// TwinCAT 3 PLC project MPS
// Title: MPS
// Company: Cosylab
// ProjectVersion: 0.1
// ProgramVersion: 3.1.4023.0
// libraries:
//   Tc2_Standard, * (Beckhoff Automation GmbH)
//   Tc2_System, * (Beckhoff Automation GmbH)
//   Tc3_Module, * (Beckhoff Automation GmbH)
// project tree:
//   DUTs/ E_2PosMonState.TcDUT, E_3PosMonState.TcDUT, E_EpicsMeasurementState.TcDUT, E_KlystronState.TcDUT, E_KlystronPPSState.TcDUT, E_MpsFault.TcDUT, E_MpsFaultSeverity.TcDUT, E_MpsState.TcDUT, E_MpsWarning.TcDUT
//   / GlobalTextList.TcGTLO, PlcTask.TcTTO, Visualization Manager.TcVMO (not stored)
//   GVLs/ CONSTANTS.TcGVL, G_EPICS.TcGVL, IO.TcGVL
//   GVLs/EpicsInterfaceDef/ ST_FaultList.TcDUT, ST_FlowMeter.TcDUT, ST_InterlockOutput.TcDUT, ST_EpicsMeasurement.TcDUT, ST_PPSInput.TcDUT, ST_StateController.TcDUT, ST_StateOutput.TcDUT, ST_TwoAxisProfileMonitor.TcDUT, ST_WarningList.TcDUT, ST_TwoAxisPopIn.TcDUT, ST_FastGateValveMonitor.TcDUT, ST_General.TcDUT, ST_LatchingAND.TcDUT, ST_Pressure.TcDUT, ST_RepetitionRate.TcDUT, ST_RtdTemperature.TcDUT, ST_ThreePositionPopIn.TcDUT, ST_TwoPositionPopIn.TcDUT
//   POUs/ FB_FlowMeter.TcPOU, FB_TwoAxisPopIn.TcPOU, FB_EpicsMeasurement.TcPOU, MpsLogicTest.TcPOU, FB_Pressure.TcPOU, FB_StateController.TcPOU, FB_TwoAxisProfileMonitor.TcPOU, FB_TwoPositionPopIn.TcPOU, FB_FastGateValveMonitor.TcPOU, FB_LatchingAND.TcPOU, FB_RepetitionRate.TcPOU, FB_ThreePositionPopIn.TcPOU, FB_Pt100.TcPOU, MAIN.TcPOU, MpsLogic.TcPOU, MpsLogicUpgrade.TcPOU, RtdReadings.TcPOU
//   VISUs/ TestGUI.TcVIS

CONFIGURATION MPS
    RESOURCE PLC ON TwinCAT3
        TASK PlcTask(INTERVAL := T#10ms, PRIORITY := 20);
        PROGRAM MAIN WITH PlcTask : MAIN;
    END_RESOURCE
END_CONFIGURATION

// ---- DUTs/E_2PosMonState.TcDUT
{attribute 'qualified_only'}
{attribute 'strict'}
TYPE E_2PosMonState :
(
	Nan := 0,
	isINSERTED := 1,
	isRETRACTED := 2,
	isMOVING := 3,
	isBROKEN := 4,
	isForcedOut := 5
);
END_TYPE

// ---- DUTs/E_3PosMonState.TcDUT
{attribute 'qualified_only'}
{attribute 'strict'}
TYPE E_3PosMonState :
(
	Nan := 0,
	isINSERTED1 := 1,
	isINSERTED2 := 2,
	isRETRACTED := 3,
	isMOVING := 4,
	isBROKEN := 5,
	isForcedOut := 6
);
END_TYPE

// ---- DUTs/E_EpicsMeasurementState.TcDUT
{attribute 'qualified_only'}
{attribute 'strict'}
TYPE E_EpicsMeasurementState :
(
	Nan := 0,
	isOkay := 1,
	isInactive := 2,
	isOutOfRange := 3,
	hasTimeout := 4
);
END_TYPE

// ---- DUTs/E_KlystronState.TcDUT
{attribute 'qualified_only'}
{attribute 'strict'}
TYPE E_KlystronState :
(
	Off := 1,
	StandbyOffRequested := 3,
	StamdbyOnRequested := 4,
	Standby := 5,
	HVOffRequested := 7,
	HVOnRequested := 8,
	HV := 9,
	TrigOffRequested := 11,
	TrigOnRequested := 12,
	Trig := 13
);
END_TYPE

// ---- DUTs/E_KlystronPPSState.TcDUT
{attribute 'qualified_only'}
{attribute 'strict'}
TYPE E_KlystronPPSState :
(
	Off := 0,
	StandbyMode := 1,
	HVMode := 2,
	TrigMode := 3,
	NoSignal := 4
);
END_TYPE

// ---- DUTs/E_MpsFault.TcDUT
{attribute 'qualified_only'}
{attribute 'strict'}
TYPE E_MpsFault :
(
	NoFault := 0,
	StandbyPPSInterlock := 10,
	StandbyMPSInterlock := 11,
	HVPPSInterlock := 20,
	HVPressureInterlock := 21,
	HVDipoleFlowInterlock := 22,
	HVDipoleThermalInterlock := 23,
	HVRFNetwork02FlowInterlock := 24,
	RFPPSInterlock := 30,
	RFMPSInterlock := 31,
	BeamSolenoidFlowInterlock := 40,
	BeamSolenoidThermalInterock := 41,
	BeamGunFlowInterlock := 42,
	BeamRFNetwork01FlowInterlock := 43,
	BeamPopInInterlock := 44
);
END_TYPE

// ---- DUTs/E_MpsFaultSeverity.TcDUT
{attribute 'qualified_only'}
{attribute 'strict'}
TYPE E_MpsFaultSeverity :
(
	NoFault := 0,
	StandbyFault := 1,
	HVFault := 2,
	RFFault := 3,
	BeamFault := 4
);
END_TYPE

// ---- DUTs/E_MpsState.TcDUT
{attribute 'qualified_only'}
{attribute 'strict'}
TYPE E_MpsState :
(
	OFF := 0,
	ExitingStandby := 1,
	EnteringStandby := 2,
	STANDBY := 3,
	ExitingHV := 4,
	EnteringHV := 5,
	HV := 6,
	SafeRoutine := 7,
	EnteringManualMode := 8,
	ManualMode := 9,
	EnteringAutomaticMode := 10,
	AutomaticMode := 11,
	SelectingEnergySetpoint := 12,
	ApplyingEnergyProfile := 13,
	LowRepRateBeamOn := 14,
	FullBeamOn := 15
);
END_TYPE

// ---- DUTs/E_MpsWarning.TcDUT
{attribute 'qualified_only'}
{attribute 'strict'}
TYPE E_MpsWarning :
(
	NoWarning := 0,
	InvalidStateRequested := 1,
	ManualModeUnreachable := 2,
	AutomaticModeUnreachable := 3
);
END_TYPE

// ---- GVLs/EpicsInterfaceDef/ST_FaultList.TcDUT
TYPE ST_FaultList :
STRUCT
	Fault_1St : E_MpsFault;
	Fault_2St : E_MpsFault;
	Fault_3St : E_MpsFault;
	Fault_4St : E_MpsFault; 
	Fault_5St : E_MpsFault; 
	Fault_6St : E_MpsFault;
	Fault_7St : E_MpsFault;
	Fault_8St : E_MpsFault;
	Fault_9St : E_MpsFault;
	Fault_10St : E_MpsFault;
END_STRUCT
END_TYPE

// ---- GVLs/EpicsInterfaceDef/ST_FlowMeter.TcDUT
TYPE ST_FlowMeter :
STRUCT
	FlowInterlockSt : BOOL;
	TemperatureInterlockSt : BOOL;
	FlowSt : LREAL;
	TemperatureSt : LREAL;
END_STRUCT
END_TYPE

// ---- GVLs/EpicsInterfaceDef/ST_InterlockOutput.TcDUT
TYPE ST_InterlockOutput :
STRUCT
	HPI_SHUTR01_OPEN_OUT : BOOL;
	HPI_SHUTR02_OPEN_OUT : BOOL;
	HPI_SOLN01_ENABLE_OUT : BOOL;
	HPI_DIP01_ENABLE_OUT : BOOL;
	HPI_KLY01_STANDBY_OUT : BOOL;
	HPI_KLY01_HVMODE_OUT : BOOL;
	HPI_KLY01_TRIGMODE_OUT : BOOL;
	HPI_KLY02_STANDBY_OUT : BOOL;
	HPI_KLY02_HVMODE_OUT : BOOL;
	HPI_KLY02_TRIGMODE_OUT : BOOL;
	
	
END_STRUCT
END_TYPE

// ---- GVLs/EpicsInterfaceDef/ST_EpicsMeasurement.TcDUT
TYPE ST_EpicsMeasurement :
STRUCT
	MeasurementValueSt : LREAL := CONSTANTS.MINIMUM_LREAL;
	MeasurementLowThresholdSt : LREAL := CONSTANTS.MINIMUM_LREAL;
	MeasurementHighThresholdSt : LREAL := CONSTANTS.MINIMUM_LREAL;
	InterlockSt : BOOL;
END_STRUCT
END_TYPE

// ---- GVLs/EpicsInterfaceDef/ST_PPSInput.TcDUT
TYPE ST_PPSInput :
STRUCT
	EnableFB_IN : BOOL;
	AllowFB_IN : BOOL;
	RFPowerFB_IN : BOOL;
	
	
END_STRUCT
END_TYPE

// ---- GVLs/EpicsInterfaceDef/ST_StateController.TcDUT
TYPE ST_StateController :
STRUCT
	StateSt : E_MpsState;
	EpicsStateSt : E_MpsState;
	TargetStateEpicsSt : E_MpsState;
	TargetStateSt : E_MpsState;
	
	Klystron01CCPSVolt01St : LREAL;
	Klystron01CCPSVolt02St : LREAL;
	Klystron01StateSt : E_KlystronState;
	Klystron01PPSStateSt : E_KlystronPPSState;
	
	Klystron02CCPSVolt01St : LREAL;
	Klystron02CCPSVolt02St : LREAL;
	Klystron02StateSt : E_KlystronState;
	Klystron02PPSStateSt : E_KlystronPPSState;
	
	FaultSeveritySt : E_MpsFaultSeverity;
	SetTargetStateSt : BOOL;
	ManualModeSt : BOOL;
	AutomaticModeSt : BOOL;
	AllowEnergyProfileLoadSt : BOOL;
	AllowLowRepRateBeamOnSt : BOOL;
	AllowFullBeamOnSt : BOOL;
END_STRUCT
END_TYPE

// ---- GVLs/EpicsInterfaceDef/ST_StateOutput.TcDUT
TYPE ST_StateOutput :
STRUCT
	StandbyEnabled_OUT : BOOL;
	HVEnabled_OUT : BOOL;
	BeamEnabled_OUT : BOOL;
	ManualModeEnabled_OUT : BOOL;
	AutomaticModeEnabled_OUT : BOOL;
END_STRUCT
END_TYPE

// ---- GVLs/EpicsInterfaceDef/ST_TwoAxisProfileMonitor.TcDUT
TYPE ST_TwoAxisProfileMonitor :
STRUCT
	//Controls
	InsertAxis1Cmd : BOOL;
	InsertAxis2Cmd : BOOL;
	RetractCmd : BOOL;
	
	//Statuses
	InsertedAxis1St : BOOL;
	InsertedAxis2St : BOOL;
	RetractedSt : BOOL;
	
	InterlockSt :BOOL;
	
	StateSt : E_3PosMonState;
	
	DisableButtonsSt :BOOL;
		
END_STRUCT
END_TYPE

// ---- GVLs/EpicsInterfaceDef/ST_WarningList.TcDUT
TYPE ST_WarningList :
STRUCT
	Warning_1St : E_MpsWarning;
	Warning_2St : E_MpsWarning;
	Warning_3St : E_MpsWarning;
	Warning_4St : E_MpsWarning; 
	Warning_5St : E_MpsWarning; 
	Warning_6St : E_MpsWarning;
	Warning_7St : E_MpsWarning;
	Warning_8St : E_MpsWarning;
	Warning_9St : E_MpsWarning;
	Warning_10St : E_MpsWarning;
END_STRUCT
END_TYPE

// ---- GVLs/EpicsInterfaceDef/ST_TwoAxisPopIn.TcDUT
TYPE ST_TwoAxisPopIn :
STRUCT
	//Controls
	Axis1_InsertPos2Cmd :BOOL;
	Axis1_RetractPos1Cmd : BOOL;
	
	Axis2_InsertPos2Cmd: BOOL;
	Axis2_RetractPos1Cmd : BOOL;
	
	//Statuses
	
	Axis1_IsInsertedPos2St : BOOL;
	Axis1_IsRetractedPos1St : BOOL;
	
	Axis2_IsInsertedPos2St : BOOL;
	Axis2_IsRetractedPos1St : BOOL;
	
	InterlockSt : BOOL;
	
	Axis1StateSt : E_2PosMonState;
	Axis2StateSt : E_2PosMonState;
	
	DisableButtonsSt :BOOL;
	
END_STRUCT
END_TYPE

// ---- GVLs/EpicsInterfaceDef/ST_FastGateValveMonitor.TcDUT
TYPE ST_FastGateValveMonitor :
STRUCT
	ClosedSt : BOOL;
	OpenSt : BOOL;
	InterlockSt : BOOL;
END_STRUCT
END_TYPE

// ---- GVLs/EpicsInterfaceDef/ST_General.TcDUT
TYPE ST_General :
STRUCT
	AcknowledgeAllCmd : BOOL;
	
END_STRUCT
END_TYPE

// ---- GVLs/EpicsInterfaceDef/ST_LatchingAND.TcDUT
TYPE ST_LatchingAND :
STRUCT
	IN_1St : BOOL;
	IN_2St : BOOL;
	IN_3St : BOOL;
	IN_4St : BOOL; 
	IN_5St : BOOL; 
	IN_6St : BOOL;
	IN_7St : BOOL;
	IN_8St : BOOL;
	IN_9St : BOOL;
	IN_10St : BOOL;
	InterlockSt : BOOL;
END_STRUCT
END_TYPE

// ---- GVLs/EpicsInterfaceDef/ST_Pressure.TcDUT
TYPE ST_Pressure :
STRUCT
	IN_1St : BOOL;
	IN_2St : BOOL;
	InterlockSt : BOOL;
END_STRUCT
END_TYPE

// ---- GVLs/EpicsInterfaceDef/ST_RepetitionRate.TcDUT
TYPE ST_RepetitionRate :
STRUCT
	RepRateAboveThresholdSt : BOOL;
	RepetitionRateHzSt : REAL;
	RepetitionRateHzThreshold : REAL;
END_STRUCT
END_TYPE

// ---- GVLs/EpicsInterfaceDef/ST_RtdTemperature.TcDUT
TYPE ST_RtdTemperature :
STRUCT
	TBL_RTD01_TEMP : REAL;
	TBL_RTD02_TEMP : REAL;
	TBL_RTD03_TEMP : REAL;
	TBL_RTD04_TEMP : REAL;
	TBL_RTD05_TEMP : REAL;
	TBL_RTD06_TEMP : REAL;
END_STRUCT
END_TYPE

// ---- GVLs/EpicsInterfaceDef/ST_ThreePositionPopIn.TcDUT
TYPE ST_ThreePositionPopIn :
STRUCT
	//Controls
	RetractPos1Cmd : BOOL;
	InsertPos2Cmd : BOOL;
	InsertPos3Cmd : BOOL;
	
	//Statuses
	RetractedPos1St : BOOL;
	InsertedPos2St : BOOL;
	InsertedPos3St : BOOL;
	
	InterlockSt :BOOL;
	
	StateSt : E_3PosMonState;
	
	DisableButtonsSt :BOOL;
		
END_STRUCT
END_TYPE

// ---- GVLs/EpicsInterfaceDef/ST_TwoPositionPopIn.TcDUT
TYPE ST_TwoPositionPopIn :
STRUCT
	//Controls
	InsertPos2Cmd : BOOL;
	RetractPos1Cmd : BOOL;
	
	//Statuses
	InsertedPos2St : BOOL;
	RetractedPos1St : BOOL;
	
	InterlockSt :BOOL;
	
	StateSt : E_2PosMonState;
		
END_STRUCT
END_TYPE

// ---- GVLs/CONSTANTS.TcGVL
{attribute 'qualified_only'}
VAR_GLOBAL CONSTANT
	MINIMUM_LREAL : LREAL := -1.7976931348623157E+308;
	MINIMUM_LREAL_THRESHOLD : LREAL := -1.7976931348623157E+300;
	APPROXIMATE_ZERO : LREAL := 0.01;
	MAX_NUMBER_OF_FAULTS : UINT := 10;
	MAX_NUMBER_OF_WARNINGS : UINT := 10;
END_VAR

// ---- GVLs/G_EPICS.TcGVL
{attribute 'qualified_only'}
VAR_GLOBAL

	RepetitionRate : ST_RepetitionRate;	
	
	StateController : ST_StateController;
	StateOutput : ST_StateOutput;

	Pressure : ST_Pressure;
	GunFlowSwitches : ST_LatchingAND;
	FastGateValve : ST_FastGateValveMonitor;
	RfNetwork01FlowSwitches : ST_LatchingAND;
	RfNetwork02FlowSwitches : ST_LatchingAND;
	SolenoidFlow : ST_LatchingAND;
	SolenoidThermalSwitches : ST_LatchingAND;
	DipoleThermalSwitches : ST_LatchingAND;
	DipoleFlow : ST_LatchingAND;
	MagnetField : ST_EpicsMeasurement;
	DipoleCurrent : ST_EpicsMeasurement; 
	
	PopIn01 : ST_ThreePositionPopIn;
	PopIn02 : ST_TwoPositionPopIn;
	PopIn03 : ST_TwoAxisPopIn;
	PopIn04 : ST_ThreePositionPopIn;
	PopIn05 : ST_TwoAxisPopIn;
	PopIn06 : ST_TwoPositionPopIn;
	
	InterlockOutput :ST_InterlockOutput;
	PPSInput : ST_PPSInput;
	
	FaultList : ST_FaultList;
	WarningList : ST_WarningList;
	
	General : ST_General;
	
	RtdTemperature	: ST_RtdTemperature;
	
	Linac1Flow : ST_LatchingAND;
	
	Linac2FlowMeter01 : ST_FlowMeter;
	Linac2FlowMeter02 : ST_FlowMeter;
	Linac2FlowMeter03 : ST_FlowMeter;
	Linac2FlowMeter04 : ST_FlowMeter;
	Linac2FlowMeter05 : ST_FlowMeter;
	Linac2Flow : ST_LatchingAND;
	
END_VAR

// ---- GVLs/IO.TcGVL
{attribute 'qualified_only'}
VAR_GLOBAL
	
BUN1_PULS01_REPRATE_IN   AT %I* : UDINT;   //   Pulse generator repetition rate
BUN1_PULS01_INHIBIT_OUT   AT %Q* : BOOL;   //Pulse generator inhibit
HPI_SHUTR01_OPEN_OUT   AT %Q* : BOOL;   //MPS Shutter, located before the HPI, opens the shutter
HPI_SHUTR02_OPEN_OUT   AT %Q* : BOOL;   //MPS Shutter, located before the HPI, opens the shutter
HPI_VGCC01_PRESSILK_IN   AT %I* : BOOL;   //   Vacuum gauge controller pressure interlock
HPI_IONP01_PRESSILK_IN   AT %I* : BOOL;   //   Ion pump controller pressure interlock
HPI_HPI01_FS1_IN   AT %I* : BOOL;   //   Photoinjector water flow
HPI_HPI01_FS2_IN   AT %I* : BOOL;   //   Photoinjector water flow
HPI_HPI01_FS3_IN   AT %I* : BOOL;   //   Photoinjector water flow
HPI_HPI01_FS4_IN   AT %I* : BOOL;   //   Photoinjector water flow
HPI_HPI01_FS5_IN   AT %I* : BOOL;   //   Photoinjector water flow
HPI_HPI01_FS6_IN   AT %I* : BOOL;   //   Photoinjector water flow
HPI_RFNET01_FS1_IN   AT %I* : BOOL;   //   RF network (loads and windows) water flow
HPI_RFNET02_FS1_IN   AT %I* : BOOL;   //   RF network (loads and windows) water flow
HPI_RFNET02_FS2_IN   AT %I* : BOOL;   //   RF network (loads and windows) water flow
HPI_RFNET02_FS3_IN   AT %I* : BOOL;   //   RF network (loads and windows) water flow
HPI_SOLN01_FS1_IN   AT %I* : BOOL;   //   Solenoid water flow
HPI_SOLN01_FS2_IN   AT %I* : BOOL;   //   Solenoid water flow
HPI_SOLN01_FS3_IN   AT %I* : BOOL;   //   Solenoid water flow
HPI_VALV01_CLOSED_IN   AT %I* : BOOL;   //   Fast acting gate valve
HPI_VALV01_OPEN_IN   AT %I* : BOOL;   //   Fast acting gate valve
HPI_KLY01_STANDBY_OUT    AT %Q* : BOOL;   //Allow Standby
HPI_KLY01_HVMODE_OUT    AT %Q* : BOOL;   //Allow HV mode
HPI_KLY01_TRIGMODE_OUT    AT %Q* : BOOL;   //Allow Trig mode
HPI_KLY02_STANDBY_OUT    AT %Q* : BOOL;   //Allow Standby
HPI_KLY02_HVMODE_OUT    AT %Q* : BOOL;   //Allow HV mode
HPI_KLY02_TRIGMODE_OUT    AT %Q* : BOOL;   //Allow Trig mode
HPI_SOLN01_ENABLE_OUT   AT %Q* : BOOL;   //Enable Solenoid PSU
HPI_DIP01_ENABLE_OUT   AT %Q* : BOOL;   //Enable Dipole PSU
HPI_SOLN01_TEMPILK1_IN   AT %I* : BOOL;   //   Solenoid thermal cutoff
HPI_SOLN01_TEMPILK2_IN   AT %I* : BOOL;   //   Solenoid thermal cutoff
HPI_SOLN01_TEMPILK3_IN   AT %I* : BOOL;   //   Solenoid thermal cutoff
DUMP_DIP01_TEMPILK1_IN   AT %I* : BOOL;   //   Dipole thermal cutoff

TBL_POPIN01_RETRACTED_POS1_IN	AT %I* : BOOL;   //Pop in 01 retracted position 1
TBL_POPIN01_INSERTED_POS2_IN	AT %I* : BOOL;   //Pop in 01 inserted position 2
TBL_POPIN01_INSERTED_POS3_IN	AT %I* : BOOL;   //Pop in 01 inserted position 3
TBL_POPIN01_INSERT_POS2_OUT	AT %Q* : BOOL;   //Insert position 2
TBL_POPIN01_INSERT_POS3_OUT	AT %Q* : BOOL;   //Insert position 3

TBL_POPIN02_RETRACTED_POS1_IN	AT %I* : BOOL;   //Pop in 02 retracted position 1
TBL_POPIN02_INSERTED_POS2_IN	AT %I* : BOOL;   //Pop in 02 inserted position 2
TBL_POPIN02_INSERT_POS2_OUT	AT %Q* : BOOL;   //Insert position 2

TBL_POPIN03_AX1_RETRACTED_POS1_IN   AT %I* : BOOL;   //   Axis1 slit retracted position 1
TBL_POPIN03_AX1_INSERTED_POS2_IN   AT %I* : BOOL;   //   Axis1 slit inserted position 2
TBL_POPIN03_AX1_INSERT_POS2_OUT   AT %Q* : BOOL;   //Axis1 insert position 2
TBL_POPIN03_AX2_RETRACTED_POS1_IN   AT %I* : BOOL;   //   Axis2 slit retracted 1
TBL_POPIN03_AX2_INSERTED_POS2_IN   AT %I* : BOOL;   //   Axis2 slit inserted 2
TBL_POPIN03_AX2_INSERT_POS2_OUT   AT %Q* : BOOL;   //Axis2 insert position 2

TBL_POPIN04_RETRACTED_POS1_IN	AT %I* : BOOL;   //Pop in 04 retracted position 1
TBL_POPIN04_INSERTED_POS2_IN	AT %I* : BOOL;   //Pop in 04 inserted position 2
TBL_POPIN04_INSERTED_POS3_IN	AT %I* : BOOL;   //Pop in 04 inserted position 3
TBL_POPIN04_INSERT_POS2_OUT	AT %Q* : BOOL;   //Insert position 2
TBL_POPIN04_INSERT_POS3_OUT	AT %Q* : BOOL;   //Insert position 3

TBL_POPIN05_AX1_RETRACTED_POS1_IN   AT %I* : BOOL;   //   Axis1 slit retracted position 1
TBL_POPIN05_AX1_INSERTED_POS2_IN   AT %I* : BOOL;  //   Axis1 slit inserted position 2
TBL_POPIN05_AX1_INSERT_POS2_OUT   AT %Q* : BOOL;   //Axis1 insert position 2
TBL_POPIN05_AX2_RETRACTED_POS1_IN   AT %I* : BOOL;   //   Axis2 slit retracted 1
TBL_POPIN05_AX2_INSERTED_POS2_IN   AT %I* : BOOL;   //   Axis2 slit inserted 2
TBL_POPIN05_AX2_INSERT_POS2_OUT   AT %Q* : BOOL;   //Axis2 insert position 2

TBL_POPIN06_RETRACTED_POS1_IN	AT %I* : BOOL;   //Pop in 06 retracted position 1
TBL_POPIN06_INSERTED_POS2_IN	AT %I* : BOOL;   //Pop in 06 inserted position 2
TBL_POPIN06_INSERT_POS2_OUT	AT %Q* : BOOL;   //Insert position 2


LIN1_FS1_IN  AT %I* : BOOL;   //   Linac 1 water flow
LIN1_FS2_IN  AT %I* : BOOL;   //   Linac 1 water flow
LIN1_FS3_IN  AT %I* : BOOL;   //   Linac 1 water flow
LIN1_FS4_IN  AT %I* : BOOL;   //   Linac 1 water flow


TBL_RTD01_TEMP   AT %I* : INT;   //   RTD temperature sensor
TBL_RTD02_TEMP   AT %I* : INT;   //   RTD temperature sensor
TBL_RTD03_TEMP   AT %I* : INT;   //   RTD temperature sensor
TBL_RTD04_TEMP   AT %I* : INT;   //   RTD temperature sensor
TBL_RTD05_TEMP   AT %I* : INT;   //   RTD temperature sensor
TBL_RTD06_TEMP   AT %I* : INT;   //   RTD temperature sensor

BUN1_IOLINK_CH01_IN AT %I* : ARRAY[0..7] OF BYTE;
BUN1_IOLINK_CH02_IN AT %I* : ARRAY[0..7] OF BYTE;
BUN1_IOLINK_CH03_IN AT %I* : ARRAY[0..7] OF BYTE;
BUN1_IOLINK_CH04_IN AT %I* : ARRAY[0..7] OF BYTE;
BUN1_IOLINK_CH05_IN AT %I* : ARRAY[0..7] OF BYTE;
BUN1_IOLINK_CH06_IN AT %I* : ARRAY[0..7] OF BYTE;



END_VAR

// ---- POUs/MAIN.TcPOU
PROGRAM MAIN
VAR
	MpsLogicUpgrade : MpsLogicUpgrade;
	RtdReadings : RtdReadings;
	//MpsLogicTest : MpsLogicTest;
	
END_VAR

//EPICS test

MpsLogicUpgrade();
RtdReadings();

//MpsLogicTest();

END_PROGRAM

// ---- POUs/MpsLogicUpgrade.TcPOU
FUNCTION_BLOCK MpsLogicUpgrade

VAR
	RepetitionRate : FB_RepetitionRate;	

	StateController : FB_StateController;
	StandbyEnabled : BOOL;
	HVEnabled : BOOL;
	HVRampDown : BOOL;
	BeamEnabled : BOOL;
	BeamRampDown : BOOL;
	ManualModeEnabled : BOOL;
	AutomaticModeEnabled : BOOL;
	
	//Interlock conditions
	StandbyInterlock :  BOOL;
	HVInterlock : BOOL;
	RFInterlock : BOOL;
	BeamInterlock : BOOL;
	
	Pressure : FB_Pressure;
	GunFlowSwitches : FB_LatchingAND;
	FastGateValve : FB_FastGateValveMonitor;
	RfNetwork01FlowSwitches : FB_LatchingAND;
	RfNetwork02FlowSwitches : FB_LatchingAND;
	SolenoidFlow : FB_LatchingAND;
	SolenoidThermalSwitches : FB_LatchingAND;
	DipoleThermalSwitches : FB_LatchingAND;
	DipoleFlow : FB_LatchingAND;
	DipoleCurrent : FB_EpicsMeasurement;
	MagnetField : FB_EpicsMeasurement;
	
	PopIn01 : FB_ThreePositionPopIn;
	PopIn02 : FB_TwoPositionPopIn;
	PopIn03 : FB_TwoAxisPopIn;
	PopIn04 : FB_ThreePositionPopIn;
	PopIn05 : FB_TwoAxisPopIn;
	PopIn06 : FB_TwoPositionPopIn;
	
	Linac1Flow : FB_LatchingAND;
	
	Linac2FlowMeter01 : FB_FlowMeter;
	Linac2FlowMeter02 : FB_FlowMeter;
	Linac2FlowMeter03 : FB_FlowMeter;
	Linac2FlowMeter04 : FB_FlowMeter;
	Linac2FlowMeter05 : FB_FlowMeter;
	Linac2Flow : FB_LatchingAND;
	
END_VAR

// Acknowledge interlocks for the FB that needs it
IF G_Epics.General.AcknowledgeAllCmd THEN
	G_Epics.General.AcknowledgeAllCmd := FALSE;
	StateController.Acknowledge();
	GunFlowSwitches.Acknowledge();
	RfNetwork01FlowSwitches.Acknowledge();
	RfNetwork02FlowSwitches.Acknowledge();
	SolenoidThermalSwitches.Acknowledge();
	DipoleThermalSwitches.Acknowledge();
	SolenoidFlow.Acknowledge();
	DipoleFlow.Acknowledge();
	DipoleCurrent.Acknowledge();
	MagnetField.Acknowledge();
	Linac1Flow.Acknowledge();
	Linac2Flow.Acknowledge();
END_IF

//======================== EPICS exchange of data =======================
StateController.Control(structure := G_Epics.StateController);

RepetitionRate.Control(structure:=G_Epics.RepetitionRate);
Pressure.Control(structure:=G_Epics.Pressure);
GunFlowSwitches.Control(structure:=G_Epics.GunFlowSwitches);
FastGateValve.Control(structure:=G_Epics.FastGateValve);
RfNetwork01FlowSwitches.Control(structure:=G_Epics.RfNetwork01FlowSwitches);
RfNetwork02FlowSwitches.Control(structure:=G_Epics.RfNetwork02FlowSwitches);
SolenoidFlow.Control(structure:=G_Epics.SolenoidFlow);
SolenoidThermalSwitches.Control(structure:=G_Epics.SolenoidThermalSwitches);
DipoleThermalSwitches.Control(structure:=G_Epics.DipoleThermalSwitches);
DipoleFlow.Control(structure:=G_Epics.DipoleFlow);
DipoleCurrent.Control(structure:=G_Epics.DipoleCurrent);
MagnetField.Control(structure:=G_Epics.MagnetField);
Linac1Flow.Control(structure:=G_Epics.Linac1Flow);
Linac2Flow.Control(structure:=G_Epics.Linac2Flow);
	

PopIn01.Control(structure:=G_Epics.PopIn01);
PopIn02.Control(structure:=G_Epics.PopIn02);
PopIn03.Control(structure:=G_Epics.PopIn03);
PopIn04.Control(structure:=G_Epics.PopIn04);
PopIn05.Control(structure:=G_Epics.PopIn05);
PopIn06.Control(structure:=G_Epics.PopIn06);

Linac2FlowMeter01.Control(structure := G_EPICS.Linac2FlowMeter01);
Linac2FlowMeter02.Control(structure := G_EPICS.Linac2FlowMeter02);
Linac2FlowMeter03.Control(structure := G_EPICS.Linac2FlowMeter03);
Linac2FlowMeter04.Control(structure := G_EPICS.Linac2FlowMeter04);
Linac2FlowMeter05.Control(structure := G_EPICS.Linac2FlowMeter05);

//Transfer interlock outputs
G_EPICS.InterlockOutput.HPI_KLY01_STANDBY_OUT:=IO.HPI_KLY01_STANDBY_OUT;
G_EPICS.InterlockOutput.HPI_KLY01_HVMODE_OUT:=IO.HPI_KLY01_HVMODE_OUT;
G_EPICS.InterlockOutput.HPI_KLY01_TRIGMODE_OUT:=IO.HPI_KLY01_TRIGMODE_OUT;
G_EPICS.InterlockOutput.HPI_KLY02_STANDBY_OUT:=IO.HPI_KLY02_STANDBY_OUT;
G_EPICS.InterlockOutput.HPI_KLY02_HVMODE_OUT:=IO.HPI_KLY02_HVMODE_OUT;
G_EPICS.InterlockOutput.HPI_KLY02_TRIGMODE_OUT:=IO.HPI_KLY02_TRIGMODE_OUT;
G_EPICS.InterlockOutput.HPI_SHUTR01_OPEN_OUT:=IO.HPI_SHUTR01_OPEN_OUT;
G_EPICS.InterlockOutput.HPI_SHUTR02_OPEN_OUT:=IO.HPI_SHUTR02_OPEN_OUT;
G_EPICS.InterlockOutput.HPI_SOLN01_ENABLE_OUT:=IO.HPI_SOLN01_ENABLE_OUT;
G_EPICS.InterlockOutput.HPI_DIP01_ENABLE_OUT:=IO.HPI_DIP01_ENABLE_OUT;

//Transfer state information
G_EPICS.StateOutput.StandbyEnabled_OUT := StandbyEnabled;
G_EPICS.StateOutput.HVEnabled_OUT := HVEnabled;
G_EPICS.StateOutput.BeamEnabled_OUT := BeamEnabled;
G_EPICS.StateOutput.ManualModeEnabled_OUT := ManualModeEnabled;
G_EPICS.StateOutput.AutomaticModeEnabled_OUT := AutomaticModeEnabled;

//Transfer faults and warnings
G_EPICS.FaultList.Fault_1St := StateController.Fault_OUT[0];
G_EPICS.FaultList.Fault_2St := StateController.Fault_OUT[1];
G_EPICS.FaultList.Fault_3St := StateController.Fault_OUT[2];
G_EPICS.FaultList.Fault_4St := StateController.Fault_OUT[3];
G_EPICS.FaultList.Fault_5St := StateController.Fault_OUT[4];
G_EPICS.FaultList.Fault_6St := StateController.Fault_OUT[5];
G_EPICS.FaultList.Fault_7St := StateController.Fault_OUT[6];
G_EPICS.FaultList.Fault_8St := StateController.Fault_OUT[7];
G_EPICS.FaultList.Fault_9St := StateController.Fault_OUT[8];
G_EPICS.FaultList.Fault_10St := StateController.Fault_OUT[9];

G_EPICS.WarningList.Warning_1St := StateController.Warning_OUT[0];
G_EPICS.WarningList.Warning_2St := StateController.Warning_OUT[1];
G_EPICS.WarningList.Warning_3St := StateController.Warning_OUT[2];
G_EPICS.WarningList.Warning_4St := StateController.Warning_OUT[3];
G_EPICS.WarningList.Warning_5St := StateController.Warning_OUT[4];
G_EPICS.WarningList.Warning_6St := StateController.Warning_OUT[5];
G_EPICS.WarningList.Warning_7St := StateController.Warning_OUT[6];
G_EPICS.WarningList.Warning_8St := StateController.Warning_OUT[7];
G_EPICS.WarningList.Warning_9St := StateController.Warning_OUT[8];
G_EPICS.WarningList.Warning_10St := StateController.Warning_OUT[9];

//======================== ELEMENT INSTANCES ======================	

//State controller
StateController(StandbyEnabled_OUT => StandbyEnabled,
				HVEnabled_OUT => HVEnabled,
				HVRampDown_OUT => HVRampDown,
				BeamEnabled_OUT => BeamEnabled,
				BeamRampDown_OUT => BeamRampDown,
				ManualModeEnabled_OUT => ManualModeEnabled,
				AutomaticModeEnabled_OUT => AutomaticModeEnabled);

//Repetition rate calculation and comparison
RepetitionRate(frequencyRaw := IO.BUN1_PULS01_REPRATE_IN, Inhibit => IO.BUN1_PULS01_INHIBIT_OUT);

//Pop ins
PopIn01(RepRate := RepetitionRate.AboveThreshold,
		Retracted_Pos1_IN := IO.TBL_POPIN01_RETRACTED_POS1_IN,
		Inserted_Pos2_IN := IO.TBL_POPIN01_INSERTED_POS2_IN,
		Inserted_Pos3_IN := IO.TBL_POPIN01_INSERTED_POS3_IN,
		Insert_Pos2_OUT => IO.TBL_POPIN01_INSERT_POS2_OUT,
		Insert_Pos3_OUT => IO.TBL_POPIN01_INSERT_POS3_OUT);

PopIn02(RepRate := RepetitionRate.AboveThreshold,
		Retracted_Pos1_IN := IO.TBL_POPIN02_RETRACTED_POS1_IN,
		Inserted_Pos2_IN := IO.TBL_POPIN02_INSERTED_POS2_IN,
		Insert_Pos2_OUT => IO.TBL_POPIN02_INSERT_POS2_OUT);

PopIn03(RepRate:=RepetitionRate.AboveThreshold,
		Axis1_RetractedPos1_IN:=IO.TBL_POPIN03_AX1_RETRACTED_POS1_IN,
		Axis1_InsertedPos2_IN:=IO.TBL_POPIN03_AX1_INSERTED_POS2_IN,
		Axis1_InsertPos2_OUT=>IO.TBL_POPIN03_AX1_INSERT_POS2_OUT,
		Axis2_RetractedPos1_IN:=IO.TBL_POPIN03_AX2_RETRACTED_POS1_IN,
		Axis2_InsertedPos2_IN:=IO.TBL_POPIN03_AX2_INSERTED_POS2_IN,
		Axis2_InsertPos2_OUT=>IO.TBL_POPIN03_AX2_INSERT_POS2_OUT);

PopIn04(RepRate := RepetitionRate.AboveThreshold,
		Retracted_Pos1_IN := IO.TBL_POPIN04_RETRACTED_POS1_IN,
		Inserted_Pos2_IN := IO.TBL_POPIN04_INSERTED_POS2_IN,
		Inserted_Pos3_IN := IO.TBL_POPIN04_INSERTED_POS3_IN,
		Insert_Pos2_OUT => IO.TBL_POPIN04_INSERT_POS2_OUT,
		Insert_Pos3_OUT => IO.TBL_POPIN04_INSERT_POS3_OUT);
	
PopIn05(RepRate:=RepetitionRate.AboveThreshold,
		Axis1_RetractedPos1_IN:=IO.TBL_POPIN05_AX1_RETRACTED_POS1_IN,
		Axis1_InsertedPos2_IN:=IO.TBL_POPIN05_AX1_INSERTED_POS2_IN,
		Axis1_InsertPos2_OUT=>IO.TBL_POPIN05_AX1_INSERT_POS2_OUT,
		Axis2_RetractedPos1_IN:=IO.TBL_POPIN05_AX2_RETRACTED_POS1_IN,
		Axis2_InsertedPos2_IN:=IO.TBL_POPIN05_AX2_INSERTED_POS2_IN,
		Axis2_InsertPos2_OUT=>IO.TBL_POPIN05_AX2_INSERT_POS2_OUT );				
		
PopIn06(RepRate := RepetitionRate.AboveThreshold,
		Retracted_Pos1_IN := IO.TBL_POPIN06_RETRACTED_POS1_IN,
		Inserted_Pos2_IN := IO.TBL_POPIN06_INSERTED_POS2_IN,
		Insert_Pos2_OUT => IO.TBL_POPIN06_INSERT_POS2_OUT);			

//Pressure interlock
Pressure(IN_1 := IO.HPI_VGCC01_PRESSILK_IN,  IN_2 := IO.HPI_IONP01_PRESSILK_IN);

//Gun flow switches interlock		 
GunFlowSwitches(IN_1 := IO.HPI_HPI01_FS1_IN,
				IN_2 := IO.HPI_HPI01_FS2_IN,
				IN_3 := IO.HPI_HPI01_FS3_IN,
				IN_4 := IO.HPI_HPI01_FS4_IN,
				//IN_5 := IO.HPI_HPI01_FS5_IN,
				IN_6 := IO.HPI_HPI01_FS6_IN );

// RF network, solenoid flow switches...		 
RfNetwork01FlowSwitches(IN_1 := IO.HPI_RFNET01_FS1_IN);
RfNetwork02FlowSwitches(IN_1 := IO.HPI_RFNET02_FS1_IN, IN_2 := IO.HPI_RFNET02_FS2_IN);// IN_3 := IO.HPI_RFNET02_FS3_IN);

SolenoidFlow(IN_1 := IO.HPI_SOLN01_FS1_IN, IN_2 := IO.HPI_SOLN01_FS2_IN, IN_3 := IO.HPI_SOLN01_FS3_IN);

SolenoidThermalSwitches(IN_1:=IO.HPI_SOLN01_TEMPILK1_IN, IN_2:=IO.HPI_SOLN01_TEMPILK2_IN, IN_3:=IO.HPI_SOLN01_TEMPILK3_IN);

DipoleThermalSwitches(IN_1:=IO.DUMP_DIP01_TEMPILK1_IN);

//HPI - Photon injector, TBL - Test beam line
DipoleFlow();//IN_1 := Linac2FlowMeter05.FlowInterlock_OUT);		

DipoleCurrent(InterlockActive_IN:=AutomaticModeEnabled, MeasurementValue_OUT => G_Epics.MagnetField.MeasurementValueSt);
MagnetField(InterlockActive_IN:=AutomaticModeEnabled, MeasurementValue_OUT => G_Epics.MagnetField.MeasurementValueSt);

FastGateValve(Closed:=IO.HPI_VALV01_CLOSED_IN, Open:=IO.HPI_VALV01_OPEN_IN);

Linac1Flow(IN_1 := IO.LIN1_FS1_IN, IN_2 := IO.LIN1_FS2_IN); // IN_3 := IO.LIN1_FS3_IN, IN_4 := IO.LIN1_FS4_IN);

Linac2FlowMeter01(FlowChannel_IN := IO.BUN1_IOLINK_CH06_IN);
Linac2FlowMeter02(FlowChannel_IN := IO.BUN1_IOLINK_CH02_IN);
Linac2FlowMeter03(FlowChannel_IN := IO.BUN1_IOLINK_CH03_IN);
Linac2FlowMeter04(FlowChannel_IN := IO.BUN1_IOLINK_CH04_IN);
Linac2FlowMeter05(FlowChannel_IN := IO.BUN1_IOLINK_CH05_IN);
Linac2Flow(IN_1 := Linac2FlowMeter01.FlowInterlock_OUT, IN_2 := Linac2FlowMeter02.FlowInterlock_OUT);
					  //IN_3 := Linac2FlowMeter03.FlowInterlock_OUT, IN_4 := Linac2FlowMeter04.FlowInterlock_OUT,
					  //IN_5 := Linac2FlowMeter05.FlowInterlock_OUT);

//======================== INTERLOCKS ======================		
//StandbyInterlock := G_EPICS.PPSInput.EnableFB_IN;
StandbyInterlock := G_EPICS.PPSInput.EnableFB_IN;
HVInterlock := StandbyInterlock AND  Pressure.Interlock AND RfNetwork02FlowSwitches.Interlock AND
			DipoleFlow.Interlock AND DipoleThermalSwitches.Interlock AND Linac1Flow.Interlock AND Linac2Flow.Interlock AND
			G_EPICS.PPSInput.AllowFB_IN;
RFInterlock := HVEnabled AND HVInterlock AND 
			G_EPICS.PPSInput.RFPowerFB_IN;
BeamInterlock := RFInterlock AND //FastGateValve.Interlock AND 
			SolenoidFlow.Interlock AND SolenoidThermalSwitches.Interlock AND GunFlowSwitches.Interlock AND
			RfNetwork01FlowSwitches.Interlock AND DipoleCurrent.Interlock AND MagnetField.Interlock;
			//Prof01.Interlock AND Prof02.Interlock AND Prof03.Interlock AND Prof04.Interlock AND Prof05.Interlock AND Prof06.Interlock


//Combining inputs for Shutter Interlock output
IO.HPI_SHUTR01_OPEN_OUT := AutomaticModeEnabled AND BeamInterlock;
IO.HPI_SHUTR02_OPEN_OUT := AutomaticModeEnabled AND BeamInterlock;

//Combining inputs for solenoid and dipole interlock output
IO.HPI_SOLN01_ENABLE_OUT := HVEnabled AND HVInterlock;
IO.HPI_DIP01_ENABLE_OUT := HVEnabled AND HVInterlock;

//Combining inputs for  Klystron interlock outputs
IO.HPI_KLY01_STANDBY_OUT := StandbyInterlock;
//IO.HPI_KLY01_STANDBY_OUT := StandbyEnabled AND StandbyInterlock;
IO.HPI_KLY01_HVMODE_OUT := (AutomaticModeEnabled OR BeamRampDown) AND BeamInterlock;
IO.HPI_KLY01_TRIGMODE_OUT := (AutomaticModeEnabled OR BeamRampDown)AND BeamInterlock;

IO.HPI_KLY02_STANDBY_OUT := StandbyInterlock;
//IO.HPI_KLY02_STANDBY_OUT := StandbyEnabled AND StandbyInterlock;
IO.HPI_KLY02_HVMODE_OUT := (HVEnabled OR HVRampDown) AND HVInterlock;
IO.HPI_KLY02_TRIGMODE_OUT := (ManualModeEnabled OR AutomaticModeEnabled OR BeamRampDown) AND RFInterlock;

IF StandbyEnabled AND NOT StandbyInterlock THEN
	IF NOT  G_EPICS.PPSInput.EnableFB_IN THEN
		StateController.AddFault(E_MpsFault.StandbyPPSInterlock, E_MpsFaultSeverity.StandbyFault);
	ELSE
		StateController.AddFault(E_MpsFault.StandbyMPSInterlock, E_MpsFaultSeverity.StandbyFault);
	END_IF
END_IF

IF HVEnabled AND NOT HVInterlock THEN
	IF NOT  G_EPICS.PPSInput.AllowFB_IN THEN
		StateController.AddFault(E_MpsFault.HVPPSInterlock, E_MpsFaultSeverity.HVFault);
	ELSIF NOT Pressure.Interlock THEN
		StateController.AddFault(E_MpsFault.HVPressureInterlock, E_MpsFaultSeverity.HVFault);
	ELSIF NOT DipoleFlow.Interlock THEN
		StateController.AddFault(E_MpsFault.HVDipoleFlowInterlock, E_MpsFaultSeverity.HVFault);
	ELSIF NOT DipoleThermalSwitches.Interlock THEN
		StateController.AddFault(E_MpsFault.HVDipoleThermalInterlock, E_MpsFaultSeverity.HVFault);
	ELSIF NOT RfNetwork02FlowSwitches.Interlock THEN
		StateController.AddFault(E_MpsFault.HVRFNetwork02FlowInterlock, E_MpsFaultSeverity.HVFault);
	END_IF
END_IF

IF (ManualModeEnabled OR AutomaticModeEnabled) AND NOT RFInterlock THEN
	IF NOT G_EPICS.PPSInput.RFPowerFB_IN THEN
		StateController.AddFault(E_MpsFault.RFPPSInterlock, E_MpsFaultSeverity.RFFault);
	ELSE
		StateController.AddFault(E_MpsFault.RFMPSInterlock, E_MpsFaultSeverity.RFFault);
	END_IF
END_IF

IF AutomaticModeEnabled AND NOT BeamInterlock THEN
	IF NOT SolenoidFlow.Interlock THEN
		StateController.AddFault(E_MpsFault.BeamSolenoidFlowInterlock, E_MpsFaultSeverity.BeamFault);
	ELSIF NOT SolenoidThermalSwitches.Interlock THEN
		StateController.AddFault(E_MpsFault.BeamSolenoidThermalInterock, E_MpsFaultSeverity.BeamFault);
	ELSIF NOT GunFlowSwitches.Interlock THEN
		StateController.AddFault(E_MpsFault.BeamGunFlowInterlock, E_MpsFaultSeverity.BeamFault);
	ELSIF NOT RFNetwork01FlowSwitches.Interlock THEN
		StateController.AddFault(E_MpsFault.BeamRFNetwork01FlowInterlock, E_MpsFaultSeverity.BeamFault);
	ELSE
		StateController.AddFault(E_MpsFault.BeamPopInInterlock, E_MpsFaultSeverity.BeamFault);
	END_IF
END_IF

END_FUNCTION_BLOCK

// ---- POUs/FB_RepetitionRate.TcPOU
FUNCTION_BLOCK FB_RepetitionRate
VAR_INPUT
	frequencyRaw : UDINT;
END_VAR
VAR_OUTPUT
	Inhibit : BOOL;
	AboveThreshold : BOOL;
END_VAR
VAR
	RepetitionRateHz : REAL;
END_VAR
VAR CONSTANT
	ScalingFactor: REAL := 100; // Scaling of raw input frequency
	Threshold : REAL := 10.0; // set this for determening AboveThreshold
END_VAR


//check the card how to scale the input and how to set the frequency in configuration
RepetitionRateHz := UDINT_TO_REAL(frequencyRaw)/ScalingFactor;

AboveThreshold := RepetitionRateHz > Threshold;

METHOD Control : BOOL
VAR_IN_OUT
	structure : ST_RepetitionRate;
END_VAR
structure.RepetitionRateHzSt := RepetitionRateHz;
structure.RepRateAboveThresholdSt := AboveThreshold;
structure.RepetitionRateHzThreshold := Threshold;
END_METHOD

END_FUNCTION_BLOCK

// ---- POUs/FB_StateController.TcPOU
FUNCTION_BLOCK FB_StateController
VAR_INPUT
END_VAR
VAR_OUTPUT
	StandbyEnabled_OUT : BOOL := FALSE;
	HVEnabled_OUT : BOOL := FALSE;
	HVRampDown_OUT : BOOL := FALSE;
	BeamEnabled_OUT : BOOL := FALSE;
	BeamRampDown_OUT : BOOL := FALSE;
	ManualModeEnabled_OUT : BOOL := FALSE;
	AutomaticModeEnabled_OUT : BOOL := FALSE;
	Fault_OUT : ARRAY[0..CONSTANTS.MAX_NUMBER_OF_FAULTS] OF E_MpsFault;
	Warning_OUT : ARRAY[0..CONSTANTS.MAX_NUMBER_OF_FAULTS] OF E_MpsWarning;
	FaultSeverity_OUT : E_MpsFaultSeverity;
	
END_VAR
VAR
	State : E_MpsState;
	TargetState : E_MpsState;
	EpicsState_RB : E_MpsState;
	
	
	NumberOfFaults : UINT := 0;
	NumberOfWarnings : UINT := 0;
	Klystron01CCPSVolt01_RB : LREAL := 0;
	Klystron01CCPSVolt02_RB : LREAL := 0;
	Klystron01State_RB : E_KlystronState;
	Klystron01PPSState_RB : E_KlystronPPSState;
	
	Klystron02State_RB : E_KlystronState;
	Klystron02CCPSVolt01_RB : LREAL := 0;
	Klystron02CCPSVolt02_RB : LREAL := 0;
	Klystron02PPSState_RB : E_KlystronPPSState;
	
	ManualMode_SET : BOOL := FALSE;
	AutomaticMode_SET : BOOL := FALSE;
	AllowEnergyProfileLoad_SET : BOOL := FALSE;
	AllowLowRepRateBeamOn_SET : BOOL := FALSE;
	AllowFullBeamOn_SET : BOOL := FALSE;
	
END_VAR

//Handles state tranistion and configures state outputs
IF State = E_MpsState.OFF THEN
	StandbyEnabled_OUT := FALSE;
	HVEnabled_OUT := FALSE;
	HVRampDown_OUT := FALSE;
	BeamEnabled_OUT := FALSE;
	BeamRampDown_OUT := FALSE;
	ManualModeEnabled_OUT := FALSE;
	AutomaticModeEnabled_OUT := FALSE;
	ManualMode_SET := FALSE;
	AutomaticMode_SET := FALSE;

//When the klystron state in any state above OFF changes to Off or StandbyOff requested
//The system will move to exiting Standby state
//The same applies for the readback of the EPICS state
ELSIF State = E_MpsState.ExitingStandby THEN
	//IF Klystron01State_RB = E_KlystronState.Off AND 
	IF TRUE THEN //Klystron02State_RB = E_KlystronState.Off THEN
		TargetState := E_MpsState.OFF;
		State := E_MpsState.OFF;
	END_IF
	StandbyEnabled_OUT := FALSE;
	HVEnabled_OUT := FALSE;
	HVRampDown_OUT := FALSE;
	BeamEnabled_OUT := FALSE;
	BeamRampDown_OUT := FALSE;
	ManualMode_SET := FALSE;
	AutomaticMode_SET := FALSE;

//Move to standby when the klystrons reach standby
ELSIF State = E_MpsState.EnteringStandby AND FaultSeverity_OUT <> E_MpsFaultSeverity.StandbyFault THEN
	StandbyEnabled_OUT := TRUE;
	IF EpicsState_RB = E_MpsState.STANDBY AND //Klystron01State_RB = E_KlystronState.Standby AND 
	    	Klystron02State_RB = E_KlystronState.Standby THEN
		State := E_MpsState.STANDBY;
	END_IF
	
ELSIF Klystron02State_RB = E_KlystronState.Off OR Klystron02State_RB = E_KlystronState.StandbyOffRequested OR
	  //Klystron01State_RB = E_KlystronState.Off OR Klystron01State_RB = E_KlystronState.StandbyOffRequested
		//OR Klystron01PPSState_RB = E_KlystronPPSState.Off OR Klystron01PPSState_RB = E_KlystronPPSState.NoSignal
		//OR Klystron02PPSState_RB = E_KlystronPPSState.Off OR Klystron02PPSState_RB = E_KlystronPPSState.NoSignal
		//EpicsState_RB = E_MpsState.OFF OR 
		EpicsState_RB = E_MpsState.ExitingStandby OR
		FaultSeverity_OUT = E_MpsFaultSeverity.StandbyFault THEN 	
	State := E_MpsState.ExitingStandby;
	
ELSIF State = E_MpsState.STANDBY THEN
	StandbyEnabled_OUT := TRUE;
	HVEnabled_OUT := FALSE;
	HVRampDown_OUT := FALSE;
	BeamEnabled_OUT := FALSE;
	BeamRampDown_OUT := FALSE;
	ManualMode_SET := FALSE;
	AutomaticMode_SET := FALSE;

//When the klystron state in any state above STANDBY changes to Standby or HV Off
//The system will move to exiting HV state
//The same applies for the readback of the EPICS state
ELSIF State = E_MpsState.ExitingHV THEN
	//IF Klystron01State_RB = E_KlystronState.Standby AND
	IF Klystron02State_RB = E_KlystronState.Standby AND 
		Klystron02CCPSVolt01_RB <= CONSTANTS.APPROXIMATE_ZERO AND Klystron02CCPSVolt02_RB <= CONSTANTS.APPROXIMATE_ZERO THEN
		State := E_MpsState.STANDBY;
		TargetState := E_MpsState.STANDBY;
	END_IF 
	HVEnabled_OUT := FALSE;
	HVRampDown_OUT := TRUE;
	BeamEnabled_OUT := FALSE;
	BeamRampDown_OUT := FALSE;
	ManualMode_SET := FALSE;
	AutomaticMode_SET := FALSE;

//Move to HV when the klystrons reach HV
ELSIF State = E_MpsState.EnteringHV AND FaultSeverity_OUT <> E_MpsFaultSeverity.HVFault THEN
	HVEnabled_OUT := TRUE;
	IF EpicsState_RB = E_MpsState.HV AND //Klystron01State_RB = E_KlystronState.Standby AND
			Klystron02State_RB = E_KlystronState.HV THEN
		State := E_MpsState.HV;
	END_IF

ELSIF Klystron02State_RB = E_KlystronState.Standby OR Klystron02State_RB = E_KlystronState.HVOffRequested
		OR EpicsState_RB = E_MpsState.STANDBY OR EpicsState_RB = E_MpsState.ExitingHV 
		OR FaultSeverity_OUT = E_MpsFaultSeverity.HVFault THEN	
	State := E_MpsState.ExitingHV;	

//Case structure manages transition to higher states
ELSIF State = E_MpsState.HV THEN
	StandbyEnabled_OUT := TRUE;
	HVEnabled_OUT := TRUE;
	HVRampDown_OUT := FALSE;
	BeamEnabled_OUT := FALSE;
	BeamRampDown_OUT := FALSE;
	
	IF ManualMode_SET = TRUE THEN
		State := E_MpsState.EnteringManualMode;
	ELSIF AutomaticMode_SET = TRUE THEN
		State := E_MpsState.EnteringAutomaticMode;
	END_IF

ELSIF State = E_MpsState.EnteringManualMode AND FaultSeverity_OUT <> E_MpsFaultSeverity.RFFault THEN
	IF (ManualMode_SET = FALSE) THEN
		State := E_MpsState.SafeRoutine;
	END_IF
	ManualModeEnabled_OUT := TRUE;
	AutomaticModeEnabled_OUT := FALSE;
	IF EpicsState_RB = E_MpsState.HV AND//Klystron01State_RB = E_KlystronState.Standby AND
			Klystron02State_RB = E_KlystronState.Trig THEN
		State := E_MpsState.ManualMode;
	END_IF
	
ELSIF State = E_MpsState.SafeRoutine THEN
	IF EpicsState_RB = E_MpsState.HV AND Klystron02State_RB = E_KlystronState.HV THEN
		State := E_MpsState.HV;
	END_IF
	BeamEnabled_OUT := FALSE;
	BeamRampDown_OUT := TRUE;
	ManualMode_SET := FALSE;
	AutomaticMode_SET := FALSE;
	ManualModeEnabled_OUT := FALSE;
	AutomaticModeEnabled_OUT := FALSE;
	
ELSIF State = E_MpsState.EnteringAutomaticMode AND FaultSeverity_OUT <> E_MpsFaultSeverity.RFFault THEN	
	IF (AutomaticMode_SET = FALSE) THEN
		State := E_MpsState.SafeRoutine;
	END_IF
	BeamEnabled_OUT := TRUE;
	BeamRampDown_OUT := FALSE;
	ManualModeEnabled_OUT := FALSE;
	AutomaticModeEnabled_OUT := TRUE;
	IF EpicsState_RB = E_MpsState.HV AND Klystron01State_RB = E_KlystronState.Trig
			AND Klystron02State_RB = E_KlystronState.Trig THEN
		State := E_MpsState.AutomaticMode;
	END_IF	

ELSIF Klystron02State_RB = E_KlystronState.HV OR Klystron02State_RB = E_KlystronState.TrigOffRequested
		OR FaultSeverity_OUT = E_MpsFaultSeverity.RFFault OR (ManualMode_SET = FALSE AND AutomaticMode_SET = FALSE) THEN	
	State := E_MpsState.SafeRoutine;	
	
ELSIF State = E_MpsState.ManualMode THEN
	BeamEnabled_OUT := FALSE;
	BeamRampDown_OUT := FALSE;
	ManualModeEnabled_OUT := TRUE;
	AutomaticModeEnabled_OUT := FALSE;
	
ELSIF Klystron01State_RB = E_KlystronState.HV OR Klystron01State_RB = E_KlystronState.TrigOffRequested
		OR Klystron02State_RB = E_KlystronState.HV OR Klystron02State_RB = E_KlystronState.TrigOffRequested
		OR FaultSeverity_OUT = E_MpsFaultSeverity.RFFault THEN	
	State := E_MpsState.SafeRoutine;
	
ELSIF State = E_MpsState.AutomaticMode THEN
	BeamEnabled_OUT := TRUE;
	BeamRampDown_OUT := FALSE;
	ManualModeEnabled_OUT := FALSE;
	AutomaticModeEnabled_OUT := TRUE;
	
END_IF

METHOD Acknowledge : BOOL
VAR_INPUT
END_VAR
VAR
	DefaultFault : ARRAY[0..CONSTANTS.MAX_NUMBER_OF_FAULTS] OF E_MpsFault;
	DefaultWarning : ARRAY[0..CONSTANTS.MAX_NUMBER_OF_WARNINGS] OF E_MpsWarning; 
END_VAR
FaultSeverity_OUT := E_MpsFaultSeverity.NoFault;
Fault_OUT := DefaultFault;
Warning_OUT := DefaultWarning;
NumberOfFaults := 0;
NumberOfWarnings := 0;
END_METHOD

METHOD AddFault : BOOL
VAR_INPUT
	Fault_IN : E_MpsFault;
	FaultType_IN : E_MpsFaultSeverity;
END_VAR
IF NumberOfFaults >= CONSTANTS.MAX_NUMBER_OF_FAULTS THEN
	NumberOfFaults := CONSTANTS.MAX_NUMBER_OF_FAULTS - 1; 
END_IF
Fault_OUT[NumberOfFaults] := Fault_IN;

//System fault severity - severity of the most severe active fault
IF FaultSeverity_OUT = E_MpsFaultSeverity.NoFault THEN
	FaultSeverity_OUT := FaultType_IN;
ELSIF FaultSeverity_OUT = E_MpsFaultSeverity.StandbyFault THEN
	FaultSeverity_OUT := E_MpsFaultSeverity.StandbyFault;
ELSIF FaultSeverity_OUT = E_MpsFaultSeverity.HVFault THEN
	IF FaultType_IN = E_MpsFaultSeverity.StandbyFault THEN
		FaultSeverity_OUT := E_MpsFaultSeverity.StandbyFault;
	END_IF
ELSIF FaultSeverity_OUT = E_MpsFaultSeverity.RFFault THEN
	IF FaultType_IN = E_MpsFaultSeverity.StandbyFault OR FaultType_IN = E_MpsFaultSeverity.HVFault THEN
		FaultSeverity_OUT := FaultType_IN;
	END_IF
ELSIF FaultSeverity_OUT = E_MpsFaultSeverity.BeamFault THEN
	IF FaultType_IN <> E_MpsFaultSeverity.NoFault THEN
		FaultSeverity_OUT := FaultType_IN;
	END_IF 
END_IF

NumberOfFaults := NumberOfFaults + 1;
END_METHOD

METHOD AddWarning : BOOL
VAR_INPUT
	Warning_IN : E_MpsWarning;
END_VAR
IF NumberOfWarnings >= CONSTANTS.MAX_NUMBER_OF_WARNINGS THEN
	NumberOfWarnings := CONSTANTS.MAX_NUMBER_OF_WARNINGS - 1; 
END_IF
Warning_OUT[NumberOfWarnings] := Warning_IN;
NumberOfWarnings := NumberOfWarnings + 1;
END_METHOD

METHOD Control : BOOL
VAR_IN_OUT
	structure : ST_StateController;
END_VAR
structure.StateSt := State;
structure.TargetStateSt := TargetState;
EpicsState_RB := structure.EpicsStateSt;
Klystron01CCPSVolt01_RB := structure.Klystron01CCPSVolt01St;
Klystron01CCPSVolt02_RB := structure.Klystron01CCPSVolt02St;
Klystron01State_RB := structure.Klystron01StateSt;
Klystron01PPSState_RB := structure.Klystron01PPSStateSt;

Klystron02CCPSVolt01_RB := structure.Klystron02CCPSVolt01St;
Klystron02CCPSVolt02_RB := structure.Klystron02CCPSVolt02St;
Klystron02State_RB := structure.Klystron02StateSt;
Klystron02PPSState_RB := structure.Klystron02PPSStateSt;
structure.FaultSeveritySt := FaultSeverity_OUT;
IF ManualMode_SET = TRUE THEN
	ManualMode_SET := structure.ManualModeSt;
	IF structure.AutomaticModeSt = TRUE THEN
		AddWarning(Warning_IN := E_MpsWarning.AutomaticModeUnreachable);
	END_IF
ELSIF AutomaticMode_SET = TRUE THEN
	AutomaticMode_SET := structure.AutomaticModeSt;
	AllowEnergyProfileLoad_SET := structure.AllowEnergyProfileLoadSt;
	AllowLowRepRateBeamOn_SET := structure.AllowLowRepRateBeamOnSt;
	AllowFullBeamOn_SET := structure.AllowFullBeamOnSt;
	IF ManualMode_SET = TRUE THEN
		AddWarning(Warning_IN := E_MpsWarning.ManualModeUnreachable);
	END_IF
ELSE	
	ManualModeEnabled_OUT := FALSE;
	AutomaticModeEnabled_OUT := FALSE;
	AllowEnergyProfileLoad_SET := FALSE;
	AllowLowRepRateBeamOn_SET := FALSE;
	AllowFullBeamOn_SET := FALSE;
	IF structure.ManualModeSt = TRUE THEN
		ManualMode_SET := TRUE;
	ELSIF structure.AutomaticModeSt = TRUE THEN
		AutomaticMode_SET := TRUE;
	END_IF
END_IF

IF structure.SetTargetStateSt THEN
	G_EPICS.StateController.SetTargetStateSt := FALSE;
	TransitionToTargetState(RequestedTargetState_IN := structure.TargetStateEpicsSt);
END_IF
END_METHOD

METHOD TransitionToTargetState : BOOL
VAR_INPUT
	RequestedTargetState_IN : E_MpsState;
END_VAR
//Reject transition to transition states
IF RequestedTargetState_IN <> E_MpsState.OFF AND RequestedTargetState_IN <> E_MpsState.STANDBY
   AND RequestedTargetState_IN <> E_MpsState.HV THEN
	AddWarning(Warning_IN := E_MpsWarning.InvalidStateRequested);
	RETURN;
END_IF

IF RequestedTargetState_IN = E_MpsState.OFF THEN
	TargetState := RequestedTargetState_IN;
	State := E_MpsState.ExitingStandby;
END_IF

IF RequestedTargetState_IN = E_MpsState.STANDBY THEN
	IF State = E_MpsState.OFF THEN
		State := E_MpsState.EnteringStandby;
		TargetState := RequestedTargetState_IN;
	ELSIF State = E_MpsState.ExitingStandby THEN
		AddWarning(Warning_IN := E_MpsWarning.InvalidStateRequested);
	ELSIF State <> E_MpsState.STANDBY AND State <> E_MpsState.EnteringStandby THEN
		State := E_MpsState.ExitingHV;
		TargetState := RequestedTargetState_IN;
	END_IF
END_IF

IF RequestedTargetState_IN = E_MpsState.HV THEN
	IF State = E_MpsState.STANDBY THEN
		State := E_MpsState.EnteringHV;
		TargetState := RequestedTargetState_IN;
	ELSIF State = E_MpsState.OFF OR State = E_MpsState.EnteringStandby
			OR State = E_MpsState.ExitingStandby OR State = E_MpsState.ExitingHV THEN
		AddWarning(Warning_IN := E_MpsWarning.InvalidStateRequested);
	ELSIF State <> E_MpsState.HV AND State <> E_MpsState.EnteringHV THEN
		State := E_MpsState.SafeRoutine;
		TargetState := RequestedTargetState_IN;
	END_IF
END_IF
END_METHOD

END_FUNCTION_BLOCK

// ---- POUs/FB_Pressure.TcPOU
FUNCTION_BLOCK FB_Pressure
VAR_INPUT
	IN_1 : BOOL :=TRUE;
	IN_2 : BOOL :=TRUE;
	
END_VAR
VAR_OUTPUT
	Interlock : BOOL;
END_VAR

Interlock := IN_1 AND IN_2;

METHOD Control : BOOL
VAR_IN_OUT
	structure : ST_Pressure;
END_VAR
structure.IN_1St := IN_1;
structure.IN_2St := IN_2;
structure.InterlockSt := Interlock;
END_METHOD

END_FUNCTION_BLOCK

// ---- POUs/FB_LatchingAND.TcPOU
FUNCTION_BLOCK FB_LatchingAND
VAR_INPUT
	IN_1 : BOOL :=TRUE;
	IN_2 : BOOL :=TRUE;
	IN_3 : BOOL :=TRUE;
	IN_4 : BOOL :=TRUE;
	IN_5 : BOOL :=TRUE;
	IN_6 : BOOL :=TRUE;
	IN_7 : BOOL :=TRUE;
	IN_8 : BOOL :=TRUE;
	IN_9 : BOOL :=TRUE;
	IN_10 : BOOL :=TRUE;
END_VAR

VAR_OUTPUT
	Interlock : BOOL;
END_VAR


IF NOT (IN_1 AND IN_2 AND IN_3 AND IN_4 AND IN_5 AND IN_6 AND IN_7 AND IN_8 AND IN_9 AND IN_10) THEN
	Interlock := FALSE;
END_IF

METHOD Acknowledge : BOOL
VAR_INPUT
END_VAR
Interlock := TRUE;
END_METHOD

METHOD Control : BOOL
VAR_IN_OUT
	structure : ST_LatchingAND;
END_VAR
structure.IN_1St:= IN_1;
structure.IN_2St:=  IN_2;
structure.IN_3St := IN_3;
structure.IN_4St  :=IN_4;
structure.IN_5St := IN_5;
structure.IN_6St:=  IN_6;
structure.IN_7St:=  IN_7;
structure.IN_8St:=  IN_8;
structure.IN_9St:=  IN_9;
structure.IN_10St:=  IN_10;
structure.InterlockSt := Interlock;
END_METHOD

END_FUNCTION_BLOCK

// ---- POUs/FB_FastGateValveMonitor.TcPOU
FUNCTION_BLOCK FB_FastGateValveMonitor
VAR_INPUT
	Closed : BOOL;
	Open : BOOL;
END_VAR
VAR_OUTPUT
	Interlock : BOOL; // MPS shutter
END_VAR
VAR
END_VAR

//Fast acting gate valve - The gate valve will get its instructions from the pressure monitoring, the MPS will only monitor

Interlock := Open AND NOT Closed;

METHOD Control : BOOL
VAR_IN_OUT
	structure : ST_FastGateValveMonitor;
END_VAR
structure.ClosedSt:=Closed;
structure.OpenSt:=Open;
structure.InterlockSt:=Interlock;
END_METHOD

END_FUNCTION_BLOCK

// ---- POUs/FB_EpicsMeasurement.TcPOU
FUNCTION_BLOCK FB_EpicsMeasurement
VAR_INPUT
	InterlockActive_IN : BOOL;
END_VAR
VAR_OUTPUT
	Interlock : BOOL;
	MeasurementValue_OUT : LREAL;
END_VAR
VAR
	MeasurementValue : LREAL;
	MeasurementLowThreshold : LREAL;
	MeasurementHighThreshold : LREAL;
	State : E_EpicsMeasurementState;
	ConnectionTimer : TON;
	Timeout : TIME := T#1.2S;
END_VAR

IF State <> E_EpicsMeasurementState.isOkay AND State <> E_EpicsMeasurementState.isInactive THEN
	Interlock := FALSE;
END_IF

IF InterlockActive_IN THEN
	IF  MeasurementValue > CONSTANTS.MINIMUM_LREAL_THRESHOLD THEN
		MeasurementValue_OUT := MeasurementValue;
		IF MeasurementValue < MeasurementLowThreshold OR MeasurementValue > MeasurementHighThreshold THEN
			State := E_EpicsMeasurementState.isOutOfRange;
		END_IF
		MeasurementValue := CONSTANTS.MINIMUM_LREAL;
		ConnectionTimer(IN := FALSE);
	ELSE
		ConnectionTimer(IN := TRUE);
	END_IF
	
	ConnectionTimer(PT := Timeout);
	
	IF ConnectionTimer.Q THEN
		State := E_EpicsMeasurementState.hasTimeout;	
	END_IF
ELSE
	State := E_EpicsMeasurementState.isInactive;
END_IF

METHOD Acknowledge : BOOL
VAR_INPUT
END_VAR
Interlock := TRUE;
State := E_EpicsMeasurementState.isOkay;
ConnectionTimer(IN := FALSE);
END_METHOD

METHOD Control : BOOL
VAR_IN_OUT
	structure : ST_EpicsMeasurement;
END_VAR
MeasurementValue := structure.MeasurementValueSt;
structure.InterlockSt := Interlock;
MeasurementLowThreshold := structure.MeasurementLowThresholdSt;
MeasurementHighThreshold := structure.MeasurementHighThresholdSt;
structure.MeasurementValueSt := CONSTANTS.MINIMUM_LREAL;
END_METHOD

END_FUNCTION_BLOCK

// ---- POUs/FB_ThreePositionPopIn.TcPOU
FUNCTION_BLOCK FB_ThreePositionPopIn
VAR_INPUT
	RepRate : BOOL;
	Retracted_Pos1_IN :BOOL;
	Inserted_Pos2_IN : BOOL;
	Inserted_Pos3_IN : BOOL;
END_VAR
VAR
	NegativeEdge : F_TRIG;
	MoveDelayTimer : TON;
	DelayBetweenMoves : TIME := T#2S;
END_VAR	

VAR_OUTPUT
	Insert_Pos2_OUT: BOOL;
	Insert_Pos3_OUT : BOOL;
	Interlock : BOOL;
	State : E_3PosMonState;
	DisableButtons : BOOL;
END_VAR

//Map the input states to enum
IF Inserted_Pos2_IN AND (NOT Inserted_Pos3_IN) AND (NOT Retracted_Pos1_IN)  THEN
	State:=E_3PosMonState.isInserted1;
ELSIF (NOT Inserted_Pos2_IN) AND Inserted_Pos3_IN AND (NOT Retracted_Pos1_IN)  THEN
	State:=E_3PosMonState.isInserted2;
ELSIF (NOT Inserted_Pos2_IN) AND (NOT Inserted_Pos3_IN) AND Retracted_Pos1_IN  THEN
	State:=E_3PosMonState.isRetracted;
ELSIF (NOT Inserted_Pos2_IN) AND (NOT Inserted_Pos3_IN) AND Retracted_Pos1_IN  THEN
	State:=E_3PosMonState.isRetracted;
ELSIF (NOT Inserted_Pos2_IN) AND (NOT Inserted_Pos3_IN) AND (NOT Retracted_Pos1_IN)  THEN
	State:=E_3PosMonState.isMoving;
	
ELSIF Inserted_Pos2_IN AND Inserted_Pos3_IN AND Retracted_Pos1_IN  THEN
	State:=E_3PosMonState.isBroken;
ELSIF NOT Inserted_Pos2_IN AND Inserted_Pos3_IN AND Retracted_Pos1_IN  THEN
	State:=E_3PosMonState.isBroken;
ELSIF Inserted_Pos2_IN AND NOT Inserted_Pos3_IN AND Retracted_Pos1_IN  THEN
	State:=E_3PosMonState.isBroken;
ELSIF Inserted_Pos2_IN AND Inserted_Pos3_IN AND NOT Retracted_Pos1_IN  THEN
	State:=E_3PosMonState.isBroken;
END_IF


//Shutter interlock behaviour
IF State = E_3PosMonState.isInserted1 AND (NOT RepRate) THEN 
	Interlock := TRUE;
ELSIF State = E_3PosMonState.isInserted2 AND (NOT RepRate) THEN 
	Interlock := TRUE;
ELSIF State = E_3PosMonState.isRetracted  THEN 
	Interlock := TRUE;
ELSE 
	Interlock := FALSE;	
END_IF


// Air solenoid behaviour
IF RepRate THEN
	Retract();	
	State := E_3PosMonState.isForcedOut;
END_IF


// Timeout in between moves

NegativeEdge(CLK:=State = E_3PosMonState.isMOVING);
MoveDelayTimer(PT:=DelayBetweenMoves);

IF NegativeEdge.Q THEN
	MoveDelayTimer(IN:=TRUE);
	DisableButtons := TRUE;
ELSIF MoveDelayTimer.Q THEN
	MoveDelayTimer(IN:=FALSE);
	DisableButtons:=FALSE;
END_IF

METHOD Control : BOOL
VAR_IN_OUT
	structure: ST_ThreePositionPopIn;
END_VAR

VAR
END_VAR
IF structure.InsertPos2Cmd THEN
	structure.InsertPos2Cmd := FALSE;
	InsertPosition1();	
END_IF

IF structure.InsertPos3Cmd THEN
	structure.InsertPos3Cmd := FALSE;
	InsertPosition2();	
END_IF

IF structure.RetractPos1Cmd THEN
	structure.RetractPos1Cmd := FALSE;
	Retract();	
END_IF

structure.StateSt := State;

structure.InsertedPos2St:=Inserted_Pos2_IN;
structure.InsertedPos3St:=Inserted_Pos3_IN;
structure.RetractedPos1St:=Retracted_Pos1_IN;

structure.InterlockSt:=Interlock;

structure.DisableButtonsSt:=DisableButtons;
END_METHOD

METHOD InsertPosition1 : BOOL
VAR_INPUT
END_VAR
IF State <> E_3PosMonState.isRetracted THEN
	RETURN;
END_IF

Insert_Pos2_OUT := TRUE;	
Insert_Pos3_OUT := FALSE;
END_METHOD

METHOD InsertPosition2 : BOOL
VAR_INPUT
END_VAR
IF State <> E_3PosMonState.isRetracted THEN
	RETURN;
END_IF

Insert_Pos2_OUT := FALSE;
Insert_Pos3_OUT := TRUE;
END_METHOD

METHOD Retract : BOOL
VAR_INPUT
END_VAR
Insert_Pos2_OUT := FALSE;	
Insert_Pos3_OUT := FALSE;
END_METHOD

END_FUNCTION_BLOCK

// ---- POUs/FB_TwoPositionPopIn.TcPOU
FUNCTION_BLOCK FB_TwoPositionPopIn
VAR_INPUT
	RepRate : BOOL; // TRUE - above RepRate Threshold
	Retracted_Pos1_IN :BOOL;
	Inserted_Pos2_IN : BOOL;
END_VAR
	
VAR_OUTPUT
	Insert_Pos2_OUT : BOOL;
	Interlock : BOOL; // MPS shutter
	State : E_2PosMonState;
	Error : BOOL; // timer expired
END_VAR

//Map the inputs to enum
IF Inserted_Pos2_IN AND Retracted_Pos1_IN THEN
	State:=E_2PosMonState.isBroken;
ELSIF Inserted_Pos2_IN AND NOT Retracted_Pos1_IN THEN
	State:=E_2PosMonState.isInserted;
ELSIF NOT Inserted_Pos2_IN AND Retracted_Pos1_IN THEN
	State:=E_2PosMonState.isRetracted;
ELSIF NOT Inserted_Pos2_IN AND NOT Retracted_Pos1_IN THEN
	State:=E_2PosMonState.isMoving;
END_IF


//Shutter interlock behaviour
IF State = E_2PosMonState.isBroken THEN //Broken
	Interlock := FALSE;
ELSIF State = E_2PosMonState.isMoving THEN //Moving
	Interlock := FALSE;
ELSIF State = E_2PosMonState.isInserted AND RepRate THEN
	Interlock := FALSE;	
ELSE 
	Interlock := TRUE;	
END_IF


// Air solenoid behaviour
IF RepRate THEN
	Retract();
	State := E_2PosMonState.isForcedOut;
END_IF

METHOD Control : BOOL
VAR_IN_OUT
	structure: ST_TwoPositionPopIn;
END_VAR

VAR
END_VAR
IF structure.InsertPos2Cmd THEN
	structure.InsertPos2Cmd := FALSE;
	Insert();	
END_IF


IF structure.RetractPos1Cmd THEN
	structure.RetractPos1Cmd := FALSE;
	Retract();	
END_IF

structure.StateSt := State;

structure.InsertedPos2St:=Inserted_Pos2_IN;
structure.RetractedPos1St:=Retracted_Pos1_IN;

structure.InterlockSt:=Interlock;
END_METHOD

METHOD Insert : BOOL
VAR_INPUT
END_VAR
IF RepRate THEN
	RETURN;
END_IF

Insert_Pos2_OUT := TRUE;
END_METHOD

METHOD Retract : BOOL
VAR_INPUT
END_VAR
Insert_Pos2_OUT := FALSE;
END_METHOD

END_FUNCTION_BLOCK

// ---- POUs/FB_TwoAxisPopIn.TcPOU
FUNCTION_BLOCK FB_TwoAxisPopIn
VAR_INPUT
	RepRate : BOOL;
	
	Axis1_InsertedPos2_IN : BOOL;
	Axis1_RetractedPos1_IN : BOOL;
	
	Axis2_InsertedPos2_IN : BOOL;
	Axis2_RetractedPos1_IN : BOOL;
END_VAR
VAR_OUTPUT
	Interlock : BOOL;
	Axis1_State : E_2PosMonState;
	Axis2_State : E_2PosMonState;
	
	Axis1_InsertPos2_OUT : BOOL;
	Axis2_InsertPos2_OUT : BOOL;
END_VAR
VAR
	Axis1 : FB_TwoPositionPopIn;
	Axis2 : FB_TwoPositionPopIn;
END_VAR

// Instances of 2 and 3 position monitor
Axis1(RepRate := RepRate, 	
			Inserted_Pos2_IN := Axis1_InsertedPos2_IN,	
			Retracted_Pos1_IN := Axis1_RetractedPos1_IN,
			Insert_Pos2_OUT => Axis1_InsertPos2_OUT,
			State => Axis1_State );
			
Axis2(RepRate := RepRate,  
		Inserted_Pos2_IN := Axis2_InsertedPos2_IN, 	
		Retracted_Pos1_IN := Axis2_RetractedPos1_IN,
		Insert_Pos2_OUT => Axis2_InsertPos2_OUT, 
		State => Axis2_State);

//Handle Horizontal -  RET Air solenoid - three way position monitor collisions

IF Axis1.State = E_2PosMonState.isBROKEN AND Axis2.State= E_2PosMonState.isINSERTED THEN 
	Axis1.Retract();
ELSIF Axis1.State = E_2PosMonState.isRETRACTED AND Axis2.State = E_2PosMonState.isBROKEN THEN 
	Axis1.Retract();
ELSIF Axis1.State = E_2PosMonState.isRETRACTED AND Axis2.State = E_2PosMonState.isINSERTED THEN 
	Axis1.Retract();
ELSIF Axis1.State = E_2PosMonState.isRETRACTED AND Axis2.State = E_2PosMonState.isMOVING THEN 
	Axis1.Retract();
ELSIF Axis1.State = E_2PosMonState.isMOVING AND Axis2.State = E_2PosMonState.isINSERTED THEN 
	Axis1.Retract();
ELSIF Axis1.State = E_2PosMonState.isMOVING AND Axis2.State = E_2PosMonState.isBROKEN THEN 
	Axis1.Retract();
END_IF
			
//Handle vertical 		two way position monitor collisions	
IF Axis1.State = E_2PosMonState.isBROKEN AND Axis2.State = E_2PosMonState.isRETRACTED THEN 
	Axis2.Retract();
ELSIF Axis1.State = E_2PosMonState.isBROKEN AND Axis2.State = E_2PosMonState.isMOVING THEN 
	Axis2.Retract();
ELSIF Axis1.State = E_2PosMonState.isINSERTED AND Axis2.State = E_2PosMonState.isBROKEN THEN 
	Axis2.Retract();
ELSIF Axis1.State = E_2PosMonState.isINSERTED AND Axis2.State = E_2PosMonState.isRETRACTED THEN 
	Axis2.Retract();
ELSIF Axis1.State = E_2PosMonState.isINSERTED AND Axis2.State = E_2PosMonState.isMOVING THEN 
	Axis2.Retract();
ELSIF Axis1.State = E_2PosMonState.isMOVING AND Axis2.State = E_2PosMonState.isRETRACTED THEN 
	Axis2.Retract();
END_IF

// Handle MPS shutter Interlock output
Interlock := Axis2.Interlock AND Axis1.Interlock AND 
			(Axis1.State = E_2PosMonState.isRETRACTED AND Axis2.State = E_2PosMonState.isINSERTED) OR
			(Axis1.State = E_2PosMonState.isRETRACTED AND Axis2.State = E_2PosMonState.isRETRACTED) OR
			(Axis1.State = E_2PosMonState.isINSERTED AND Axis2.State= E_2PosMonState.isRETRACTED);

METHOD Control : BOOL
VAR_IN_OUT
	structure : ST_TwoAxisPopIn;
END_VAR
//Commands
IF structure.Axis1_InsertPos2Cmd THEN
	structure.Axis1_InsertPos2Cmd:=FALSE;
	InsertAxis1();
END_IF

IF structure.Axis1_RetractPos1Cmd THEN
	structure.Axis1_RetractPos1Cmd:=FALSE;
	RetractAxis1();
END_IF

IF structure.Axis2_InsertPos2Cmd THEN
	structure.Axis2_InsertPos2Cmd:=FALSE;
	InsertAxis2();
END_IF

IF structure.Axis2_RetractPos1Cmd THEN
	structure.Axis2_RetractPos1Cmd:=FALSE;
	RetractAxis2();
END_IF

//Statuses

structure.Axis1_IsInsertedPos2St:=Axis1.Inserted_Pos2_IN;
structure.Axis1_IsRetractedPos1St:=Axis1.Retracted_Pos1_IN;

structure.Axis2_IsInsertedPos2St:=Axis2.Inserted_Pos2_IN;
structure.Axis2_IsRetractedPos1St:=Axis2.Retracted_Pos1_IN;

structure.InterlockSt:=Interlock;

structure.Axis1StateSt:=Axis1_State;
structure.Axis2StateSt:=Axis2_State;
END_METHOD

METHOD InsertAxis1 : BOOL
VAR_INPUT
END_VAR
IF Axis1.State = E_3PosMonState.isBROKEN AND Axis2.State= E_2PosMonState.isINSERTED THEN 
	RETURN;
ELSIF Axis1.State = E_3PosMonState.isRETRACTED AND Axis2.State = E_2PosMonState.isBROKEN THEN 
	RETURN;
ELSIF Axis1.State = E_3PosMonState.isRETRACTED AND Axis2.State = E_2PosMonState.isINSERTED THEN 
	RETURN;
ELSIF Axis1.State = E_3PosMonState.isRETRACTED AND Axis2.State = E_2PosMonState.isMOVING THEN 
	RETURN;
ELSIF Axis1.State = E_3PosMonState.isMOVING AND Axis2.State = E_2PosMonState.isINSERTED THEN 
	RETURN;
ELSIF Axis1.State = E_3PosMonState.isMOVING AND Axis2.State = E_2PosMonState.isBROKEN THEN 
	RETURN;
END_IF

Axis1.Insert();
END_METHOD

METHOD InsertAxis2 : BOOL
VAR_INPUT
END_VAR
IF Axis1.State = E_2PosMonState.isBROKEN AND Axis2.State= E_2PosMonState.isRETRACTED THEN 
	RETURN;
ELSIF Axis1.State = E_2PosMonState.isBROKEN AND Axis2.State= E_2PosMonState.isMOVING THEN 
	RETURN;
ELSIF Axis1.State = E_2PosMonState.isINSERTED AND Axis2.State = E_2PosMonState.isBROKEN THEN 
	RETURN;
ELSIF Axis1.State = E_2PosMonState.isINSERTED AND Axis2.State = E_2PosMonState.isRETRACTED THEN 
	RETURN;
ELSIF Axis1.State = E_2PosMonState.isINSERTED AND Axis2.State = E_2PosMonState.isMOVING THEN 
	RETURN;
ELSIF Axis1.State = E_3PosMonState.isMOVING AND Axis2.State = E_2PosMonState.isRETRACTED THEN 
	RETURN;
END_IF

Axis2.Insert();
END_METHOD

METHOD RetractAxis1 : BOOL
VAR_INPUT
END_VAR
Axis1.Retract();
END_METHOD

METHOD RetractAxis2 : BOOL
VAR_INPUT
END_VAR
Axis2.Retract();
END_METHOD

END_FUNCTION_BLOCK

// ---- POUs/FB_FlowMeter.TcPOU
FUNCTION_BLOCK FB_FlowMeter
VAR_INPUT
	FlowChannel_IN : ARRAY[0..7] OF BYTE;
END_VAR
VAR_OUTPUT
	FlowInterlock_OUT : BOOL;
	TemperatureInterlock_OUT : BOOL;
	Flow_OUT : LREAL;
	Temperature_OUT : LREAL;
END_VAR
VAR
	FlowRaw : INT;
	TemperatureRaw : INT;
END_VAR

VAR CONSTANT
	FLOW_COEF : LREAL := 0.04;
	TEMP_COEF : LREAL := 0.1;
END_VAR

FlowInterlock_OUT := FlowChannel_IN[5].0;
TemperatureInterlock_OUT := FlowChannel_IN[5].1;
TemperatureRaw := BYTE_TO_INT(FlowChannel_IN[2]) * 256 + BYTE_TO_INT(FlowChannel_IN[3]);
FlowRaw := BYTE_TO_INT(FlowChannel_IN[0]) * 256 + BYTE_TO_INT(FlowChannel_IN[1]);
Temperature_OUT := INT_TO_LREAL(TemperatureRaw) * TEMP_COEF;
Flow_OUT := INT_TO_LREAL(FlowRaw) * FLOW_COEF;

METHOD Control : BOOL
VAR_IN_OUT
	structure : ST_FlowMeter;
END_VAR
structure.FlowInterlockSt := FlowInterlock_OUT;
structure.TemperatureInterlockSt := TemperatureInterlock_OUT;
structure.FlowSt := Flow_OUT;
structure.TemperatureSt := Temperature_OUT;
END_METHOD

END_FUNCTION_BLOCK

// ---- POUs/RtdReadings.TcPOU
FUNCTION_BLOCK RtdReadings

VAR
	Rtd01 : FB_Pt100;
	Rtd02 : FB_Pt100;
	Rtd03 : FB_Pt100;
	Rtd04 : FB_Pt100;
	Rtd05 : FB_Pt100;
	Rtd06 : FB_Pt100;
END_VAR

//Instances of PT100, temperature measurement
Rtd01(Raw := IO.TBL_RTD01_TEMP,TempFaranheit =>G_Epics.RtdTemperature.TBL_RTD01_TEMP);
Rtd02(Raw := IO.TBL_RTD02_TEMP,TempFaranheit =>G_Epics.RtdTemperature.TBL_RTD02_TEMP);
Rtd03(Raw := IO.TBL_RTD03_TEMP,TempFaranheit =>G_Epics.RtdTemperature.TBL_RTD03_TEMP);
Rtd04(Raw := IO.TBL_RTD04_TEMP,TempFaranheit =>G_Epics.RtdTemperature.TBL_RTD04_TEMP);
Rtd05(Raw := IO.TBL_RTD05_TEMP,TempFaranheit =>G_Epics.RtdTemperature.TBL_RTD05_TEMP);
Rtd06(Raw := IO.TBL_RTD06_TEMP,TempFaranheit =>G_Epics.RtdTemperature.TBL_RTD06_TEMP);

END_FUNCTION_BLOCK

// ---- POUs/FB_Pt100.TcPOU
FUNCTION_BLOCK FB_Pt100
VAR_INPUT
	Raw : INT;
END_VAR
VAR_OUTPUT
	TempCelsius : REAL;
	TempFaranheit : REAL;
END_VAR

// Card settings: 3-wire, 0,1°C precision, pt100

TempCelsius:= Raw/10;
TempFaranheit := (TempCelsius*9/5)+32;

END_FUNCTION_BLOCK

// ---- POUs/MpsLogicTest.TcPOU
FUNCTION_BLOCK MpsLogicTest
VAR
	StateController : FB_StateController;
	StandbyEnabled : BOOL;
	HVEnabled : BOOL;
	BeamEnabled : BOOL;
	ManualModeEnabled : BOOL;
	AutomaticModeEnabled : BOOL;
	
	MpsStateList : ARRAY[0..17] OF E_MpsState := [E_MpsState.OFF, E_MpsState.STANDBY, E_MpsState.EnteringStandby, E_MpsState.ExitingStandby, E_MpsState.HV, E_MpsState.EnteringHV, E_MpsState.ExitingHV, E_MpsState.SafeRoutine, E_MpsState.ManualMode, E_MpsState.EnteringManualMode, E_MpsState.SelectingEnergySetpoint, E_MpsState.ApplyingEnergyProfile, E_MpsState.LowRepRateBeamOn, E_MpsState.FullBeamOn];
	MpsSelectedTargetState : INT;
	MpsSelectedEPICSState : INT;
	KlystronStateList : ARRAY[0..9] OF E_KlystronState := [E_KlystronState.Off, E_KlystronState.StandbyOffRequested, E_KlystronState.StamdbyOnRequested, E_KlystronState.Standby, E_KlystronState.HVOffRequested, E_KlystronState.HVOnRequested, E_KlystronState.HV, E_KlystronState.TrigOffRequested, E_KlystronState.TrigOnRequested, E_KlystronState.Trig];
	
	SetTargetStateEPICS : BOOL;
	SetEPICSState : BOOL;
END_VAR

IF G_Epics.General.AcknowledgeAllCmd THEN
	G_Epics.General.AcknowledgeAllCmd := FALSE;
END_IF


//======================== EPICS exchange of data =================
StateController.Control(structure := G_Epics.StateController);

//======================== ELEMENT INSTANCES ======================	
StateController(StandbyEnabled_OUT => StandbyEnabled,
				HVEnabled_OUT => HVEnabled,
				BeamEnabled_OUT => BeamEnabled);

END_FUNCTION_BLOCK

// ---- POUs/FB_TwoAxisProfileMonitor.TcPOU
FUNCTION_BLOCK FB_TwoAxisProfileMonitor
VAR_INPUT
	RepRate : BOOL;
	Retracted_IN :BOOL;
	Inserted_Axis_1_IN : BOOL;
	Inserted_Axis_2_IN : BOOL;
END_VAR
VAR
	NegativeEdge : F_TRIG;
	MoveDelayTimer : TON;
	DelayBetweenMoves : TIME := T#2S;
END_VAR	

VAR_OUTPUT
	Insert_Axis_1_OUT: BOOL;
	Insert_Axis_2_OUT : BOOL;
	Interlock : BOOL;
	State : E_3PosMonState;
	DisableButtons : BOOL;
END_VAR

//Map the input states to enum
IF Inserted_Axis_1_IN AND (NOT Inserted_Axis_2_IN) AND (NOT Retracted_IN)  THEN
	State:=E_3PosMonState.isInserted1;
ELSIF (NOT Inserted_Axis_1_IN) AND Inserted_Axis_2_IN AND (NOT Retracted_IN)  THEN
	State:=E_3PosMonState.isInserted2;
ELSIF (NOT Inserted_Axis_1_IN) AND (NOT Inserted_Axis_2_IN) AND Retracted_IN  THEN
	State:=E_3PosMonState.isRetracted;
ELSIF (NOT Inserted_Axis_1_IN) AND (NOT Inserted_Axis_2_IN) AND Retracted_IN  THEN
	State:=E_3PosMonState.isRetracted;
ELSIF (NOT Inserted_Axis_1_IN) AND (NOT Inserted_Axis_2_IN) AND (NOT Retracted_IN)  THEN
	State:=E_3PosMonState.isMoving;
	
ELSIF Inserted_Axis_1_IN AND Inserted_Axis_2_IN AND Retracted_IN  THEN
	State:=E_3PosMonState.isBroken;
ELSIF NOT Inserted_Axis_1_IN AND Inserted_Axis_2_IN AND Retracted_IN  THEN
	State:=E_3PosMonState.isBroken;
ELSIF Inserted_Axis_1_IN AND NOT Inserted_Axis_2_IN AND Retracted_IN  THEN
	State:=E_3PosMonState.isBroken;
ELSIF Inserted_Axis_1_IN AND Inserted_Axis_2_IN AND NOT Retracted_IN  THEN
	State:=E_3PosMonState.isBroken;
END_IF


//Shutter interlock behaviour
IF State = E_3PosMonState.isInserted1 AND (NOT RepRate) THEN 
	Interlock := TRUE;
ELSIF State = E_3PosMonState.isInserted2 AND (NOT RepRate) THEN 
	Interlock := TRUE;
ELSIF State = E_3PosMonState.isRetracted  THEN 
	Interlock := TRUE;
ELSE 
	Interlock := FALSE;	
END_IF


// Air solenoid behaviour
IF RepRate THEN
	Retract();	
	State := E_3PosMonState.isForcedOut;
END_IF


// Timeout in between moves

NegativeEdge(CLK:=State = E_3PosMonState.isMOVING);
MoveDelayTimer(PT:=DelayBetweenMoves);

IF NegativeEdge.Q THEN
	MoveDelayTimer(IN:=TRUE);
	DisableButtons := TRUE;
ELSIF MoveDelayTimer.Q THEN
	MoveDelayTimer(IN:=FALSE);
	DisableButtons:=FALSE;
END_IF

METHOD Control : BOOL
VAR_IN_OUT
	structure: ST_ThreePositionPopIn;
END_VAR

VAR
END_VAR
IF structure.InsertPos2Cmd THEN
	structure.InsertPos2Cmd := FALSE;
	InsertAxis1();	
END_IF

IF structure.InsertPos3Cmd THEN
	structure.InsertPos3Cmd := FALSE;
	InsertAxis2();	
END_IF

IF structure.RetractPos1Cmd THEN
	structure.RetractPos1Cmd := FALSE;
	Retract();	
END_IF

structure.StateSt := State;

structure.InsertedPos2St:=Inserted_Axis_1_IN;
structure.InsertedPos3St:=Inserted_Axis_2_IN;
structure.RetractedPos1St:=Retracted_IN;

structure.InterlockSt:=Interlock;

structure.DisableButtonsSt:=DisableButtons;
END_METHOD

METHOD InsertAxis1 : BOOL
VAR_INPUT
END_VAR
IF State <> E_3PosMonState.isRetracted THEN
	RETURN;
END_IF

Insert_Axis_1_OUT := TRUE;	
Insert_Axis_2_OUT := FALSE;
END_METHOD

METHOD InsertAxis2 : BOOL
VAR_INPUT
END_VAR
IF State <> E_3PosMonState.isRetracted THEN
	RETURN;
END_IF

Insert_Axis_1_OUT := FALSE;
Insert_Axis_2_OUT := TRUE;
END_METHOD

METHOD Retract : BOOL
VAR_INPUT
END_VAR
Insert_Axis_1_OUT := FALSE;	
Insert_Axis_2_OUT := FALSE;
END_METHOD

END_FUNCTION_BLOCK

// ---- POUs/MpsLogic.TcPOU
FUNCTION_BLOCK MpsLogic

VAR
	RepetitionRate : FB_RepetitionRate;	

	Pressure : FB_Pressure;
	GunFlowSwitches : FB_LatchingAND;
	FastGateValve : FB_FastGateValveMonitor;
	RfNetworkFlowSwitches : FB_LatchingAND;
	SolenoidFlow : FB_LatchingAND;
	SolenoidThermalSwitches : FB_LatchingAND;
	DipoleFlow : FB_LatchingAND;
	
	DipoleCurrent : FB_EpicsMeasurement;
	MagnetField : FB_EpicsMeasurement;
	
	Prof01 : FB_TwoAxisPopIn;
	Prof02 : FB_TwoAxisPopIn;
	
	
END_VAR

// Acknowledge interlocks for the FB that needs it
IF G_Epics.General.AcknowledgeAllCmd THEN
	G_Epics.General.AcknowledgeAllCmd := FALSE;
	GunFlowSwitches.Acknowledge();
	RfNetworkFlowSwitches.Acknowledge();
	SolenoidThermalSwitches.Acknowledge();
	SolenoidFlow.Acknowledge();
	//DipoleFlow.Acknowledge();
	DipoleCurrent.Acknowledge();
	//MagnetField.Acknowledge();
END_IF

//======================== EPICS exchange of data ======================	
RepetitionRate.Control(structure:=G_Epics.RepetitionRate);
Pressure.Control(structure:=G_Epics.Pressure);
GunFlowSwitches.Control(structure:=G_Epics.GunFlowSwitches);
FastGateValve.Control(structure:=G_Epics.FastGateValve);
RfNetworkFlowSwitches.Control(structure:=G_Epics.RfNetworkFlowSwitches);
SolenoidFlow.Control(structure:=G_Epics.SolenoidFlow);
SolenoidThermalSwitches.Control(structure:=G_Epics.SolenoidThermalSwitches);
//DipoleFlow.Control(structure:=G_Epics.DipoleFlow);
DipoleCurrent.Control(structure:=G_Epics.DipoleCurrent);
//MagnetField.Control(structure:=G_Epics.MagnetField);
	

Prof01.Control(structure:=G_Epics.PopIn03);
Prof02.Control(structure:=G_Epics.PopIn05);


G_EPICS.InterlockOutput.HPI_KLY01_STANDBY_OUT:=IO.HPI_KLY01_STANDBY_OUT;
G_EPICS.InterlockOutput.HPI_KLY01_HVMODE_OUT:=IO.HPI_KLY01_HVMODE_OUT;
G_EPICS.InterlockOutput.HPI_KLY01_TRIGMODE_OUT:=IO.HPI_KLY01_TRIGMODE_OUT;
G_EPICS.InterlockOutput.HPI_SHUTR01_OPEN_OUT:=IO.HPI_SHUTR01_OPEN_OUT;
G_EPICS.InterlockOutput.HPI_SOLN01_ENABLE_OUT:=IO.HPI_SOLN01_ENABLE_OUT;

//======================== ELEMENT INSTANCES ======================	

//Repetition rate calculation and comparison
RepetitionRate(frequencyRaw := IO.BUN1_PULS01_REPRATE_IN, Inhibit => IO.BUN1_PULS01_INHIBIT_OUT);

//Profile monitors and eslits instances	
Prof01(RepRate:=RepetitionRate.AboveThreshold,
		Axis1_RetractedPos1_IN:=IO.TBL_POPIN03_AX1_RETRACTED_POS1_IN,
		Axis1_InsertedPos2_IN:=IO.TBL_POPIN03_AX1_INSERTED_POS2_IN,
		Axis1_InsertPos2_OUT=>IO.TBL_POPIN03_AX1_INSERT_POS2_OUT,
		Axis2_RetractedPos1_IN:=IO.TBL_POPIN03_AX2_RETRACTED_POS1_IN,
		Axis2_InsertedPos2_IN:=IO.TBL_POPIN03_AX2_INSERTED_POS2_IN,
		Axis2_InsertPos2_OUT=>IO.TBL_PROF01_V_INSERT_OUT );
		
Prof02(RepRate:=RepetitionRate.AboveThreshold,
		Axis1_RetractedPos1_IN:=IO.TBL_POPIN05_AX1_RETRACTED_POS1_IN,
		Axis1_InsertedPos2_IN:=IO.TBL_POPIN05_AX1_INSERTED_POS2_IN,
		Axis1_InsertPos2_OUT=>IO.TBL_POPIN05_AX1_INSERT_POS2_OUT,
		Axis2_RetractedPos1_IN:=IO.TBL_POPIN05_AX2_RETRACTED_POS1_IN,
		Axis2_InsertedPos2_IN:=IO.TBL_POPIN05_AX2_INSERTED_POS2_IN,
		Axis2_InsertPos2_OUT=>IO.TBL_POPIN05_AX2_INSERT_POS2_OUT );				

//Pressure interlock
Pressure(IN_1 := IO.HPI_VGCC01_PRESSILK_IN,  IN_2 := IO.HPI_IONP01_PRESSILK_IN);

//Gun flow switches interlock		 
GunFlowSwitches(IN_1 := IO.HPI_HPI01_FS1_IN,
				IN_2 := IO.HPI_HPI01_FS2_IN,
				IN_3 := IO.HPI_HPI01_FS3_IN,
				IN_4 := IO.HPI_HPI01_FS4_IN,
				IN_5 := IO.HPI_HPI01_FS5_IN,
				IN_6 := IO.HPI_HPI01_FS6_IN );

// RF network, solenoid flow switches...		 
RfNetworkFlowSwitches(IN_1 := IO.HPI_RFNET01_FS_IN, IN_2 := IO.HPI_RFNET02_FS_IN, IN_3 := IO.HPI_RFNET03_FS_IN);

SolenoidFlow(IN_1 := IO.HPI_SOLN01_FS1_IN, IN_2 := IO.HPI_SOLN01_FS2_IN, IN_3 := IO.HPI_SOLN01_FS3_IN);

SolenoidThermalSwitches(IN_1:=IO.HPI_SOLN01_TEMPILK1_IN, IN_2:=IO.HPI_SOLN01_TEMPILK2_IN, IN_3:=IO.HPI_SOLN01_TEMPILK3_IN);

//What does HPI stand for?? Maybe Hardware Protection Interlock?
//DipoleFlow(IN = IO.HPI_DPM01_FS1_IN);		

MagnetField();
		
FastGateValve(Closed:=IO.HPI_VALV01_CLOSED_IN, Open:=IO.HPI_VALV01_OPEN_IN);		

//======================== INTERLOCKS ======================		
		
//Combining inputs for Shutter Interlock output
IO.HPI_SHUTR01_OPEN_OUT:=Pressure.Interlock AND FastGateValve.Interlock AND SolenoidFlow.Interlock AND 
						SolenoidThermalSwitches.Interlock AND DipoleFlow.Interlock AND IO.HPI_SOLN01_ENABLE_OUT AND GunFlowSwitches.Interlock AND
						Prof01.Interlock AND Prof02.Interlock AND RfNetworkFlowSwitches.Interlock;

//Combining inputs for  Solenoid interlock output
IO.HPI_SOLN01_ENABLE_OUT:=SolenoidFlow.Interlock AND SolenoidThermalSwitches.Interlock;

//Combining inputs for  Klystron interlock outputs
IO.HPI_KLY01_STANDBY_OUT := TRUE;
IO.HPI_KLY01_HVMODE_OUT :=Pressure.Interlock AND SolenoidFlow.Interlock AND GunFlowSwitches.Interlock AND 
						SolenoidThermalSwitches.Interlock AND DipoleFlow.Interlock AND RfNetworkFlowSwitches.Interlock;
IO.HPI_KLY01_TRIGMODE_OUT := IO.HPI_KLY01_HVMODE_OUT;

END_FUNCTION_BLOCK

// ---- GlobalTextList.TcGTLO
TEXTLIST GlobalTextList
  909 = 'Acknowledge ALL Faults'
  304 = 'Beam Enabled'
  548 = 'EPICS State'
  208 = 'Fault Type: %s'
  41 = 'Faults:'
  574 = 'HV Enabled'
  618 = 'Klystron 1 State'
  312 = 'Klystron State: %s'
  339 = 'Requested Target State'
  993 = 'Set EPICS state'
  557 = 'Set Target State'
  89 = 'Standby Enabled'
  113 = 'State: %s'
  218 = 'Target State: %s'
  803 = 'Warnings:'
END_TEXTLIST

// ---- VISUs/TestGUI.TcVIS
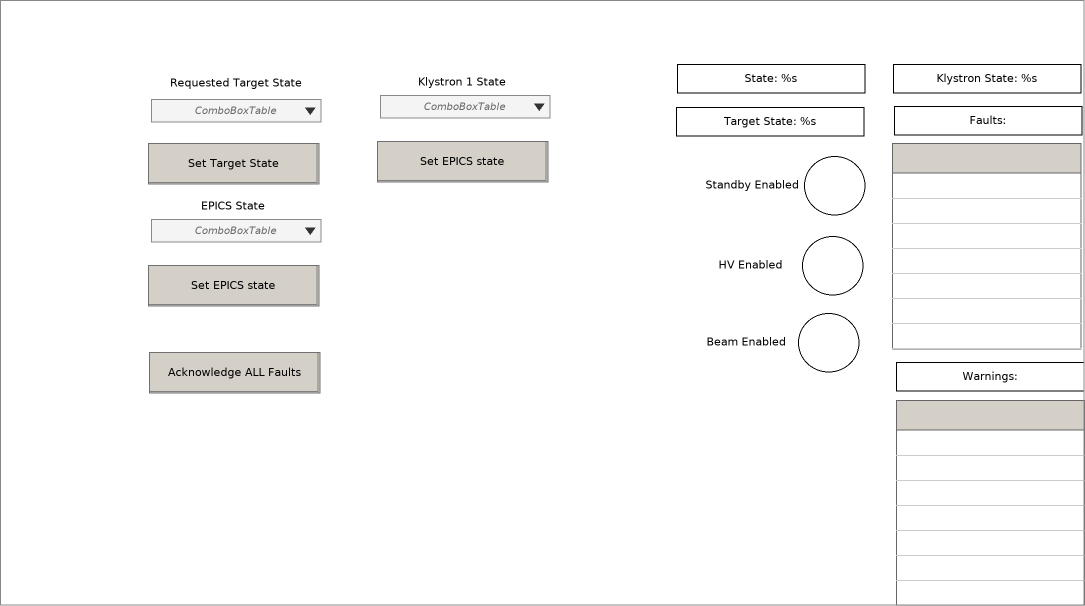
VISUALIZATION TestGUI  // 1085x606
    Button (148,143 171x41), "Set Target State"
        toggle MAIN.MpsLogicTest.SetTargetStateEPICS
    ComboBoxTable (151,99 170x23), variable: MAIN.MpsLogicTest.MpsSelectedTargetState, data array: MAIN.MpsLogicTest.MpsStateList
        p3854506369: MAIN.MpsLogicTest.MpsStateList[INDEX]
    Rectangle (677,64 188x29), "State: %s", text variable: MAIN.MpsLogicTest.StateController.State
    Ellipse (804,156 61x59), colour toggle: MAIN.MpsLogicTest.StandbyEnabled
    Label (703,170 99x30), "Standby Enabled"
    Ellipse (802,236 61x59), colour toggle: MAIN.MpsLogicTest.HVEnabled
    Label (701,250 99x30), "HV Enabled"
    Ellipse (798,313 61x59), colour toggle: MAIN.MpsLogicTest.BeamEnabled
    Label (697,327 99x30), "Beam Enabled"
    Rectangle (676,107 188x29), "Target State: %s", text variable: MAIN.MpsLogicTest.StateController.TargetState
    Rectangle (893,64 188x29), "Klystron State: %s", text variable: MAIN.MpsLogicTest.StateController.Klystron01State_RB
    Label (152,68 168x30), "Requested Target State"
    ComboBoxTable (151,219 170x23), variable: MAIN.MpsLogicTest.MpsSelectedEPICSState, data array: MAIN.MpsLogicTest.MpsStateList
        p3854506369: MAIN.MpsLogicTest.MpsStateList[INDEX]
    Label (148,191 170x30), "EPICS State"
    Button (148,265 171x41), "Set EPICS state"
        toggle MAIN.MpsLogicTest.SetEPICSState
    Table (892,143 189x206), data array: MAIN.MpsLogicTest.StateController.Fault_OUT
        p3854506369: MAIN.MpsLogicTest.StateController.Fault_OUT[INDEX]
        p2232123230: MAIN.MpsLogicTest.StateController.Fault[INDEX]
        p2685023577: MAIN.MpsLogicTest.StateController.Fault_OUT_OUT[INDEX]
    Table (896,400 189x206), data array: MAIN.MpsLogicTest.StateController.Warning_OUT
        p3854506369: MAIN.MpsLogicTest.StateController.Warning_OUT[INDEX]
        p2232123230: MAIN.MpsLogicTest.StateController.Warning[INDEX]
        p2685023577: MAIN.MpsLogicTest.StateController.Warning_OUT_OUT[INDEX]
    Rectangle (894,106 188x29), "Faults:"
    Rectangle (896,362 188x29), "Warnings:"
    Button (149,352 171x41), "Acknowledge ALL Faults"
        toggle G_Epics.General.AcknowledgeAllCmd
    ComboBoxTable (380,95 170x23), variable: MAIN.MpsLogicTest.StateController.Klystron01State_RB, data array: MAIN.MpsLogicTest.MpsStateList
        p3854506369: MAIN.MpsLogicTest.MpsStateList[INDEX]
    Label (377,67 170x30), "Klystron 1 State"
    Button (377,141 171x41), "Set EPICS state"
        toggle MAIN.MpsLogicTest.SetEPICSState
END_VISUALIZATION
